LIN {X 0.076,Y -557.564,Z 1031.331,A 0.000,B 0.000,C 90.000,E1 95.625} C_DIS
LIN {X -0.086,Y -558.588,Z 1031.325,A 0.000,B 0.000,C 90.000,E1 94.531} C_DIS
LIN {X -0.162,Y -559.455,Z 1031.318,A 0.000,B 0.000,C 90.000,E1 93.151} C_DIS
LIN {X 0.192,Y -560.065,Z 1031.311,A 0.000,B 0.000,C 90.000,E1 92.007} C_DIS
LIN {X -0.259,Y -560.817,Z 1031.301,A 0.000,B 0.000,C 90.000,E1 90.115} C_DIS
LIN {X -0.131,Y -561.493,Z 1031.290,A 0.000,B 0.000,C 90.000,E1 88.165} C_DIS
LIN {X -0.179,Y -561.938,Z 1031.282,A 0.000,B 0.000,C 90.000,E1 86.788} C_DIS
LIN {X -0.001,Y -562.460,Z 1031.271,A 0.000,B 0.000,C 90.000,E1 84.837} C_DIS
LIN {X 0.054,Y -562.784,Z 1031.264,A 0.000,B 0.000,C 90.000,E1 83.451} C_DIS
LIN {X 0.026,Y -563.425,Z 1031.250,A 0.000,B 0.000,C 90.000,E1 80.971} C_DIS
LIN {X -0.056,Y -564.060,Z 1031.239,A 0.000,B 0.000,C 90.000,E1 79.050} C_DIS
LIN {X -0.009,Y -565.007,Z 1031.229,A 0.000,B 0.000,C 90.000,E1 77.117} C_DIS
LIN {X -0.145,Y -565.830,Z 1031.221,A 0.000,B 0.000,C 90.000,E1 75.755} C_DIS
LIN {X 0.008,Y -567.631,Z 1031.207,A 0.000,B 0.000,C 90.000,E1 73.268} C_DIS
LIN {X 0.206,Y -569.135,Z 1031.196,A 0.000,B 0.000,C 90.000,E1 71.329} C_DIS
LIN {X -0.249,Y -570.167,Z 1031.189,A 0.000,B 0.000,C 90.000,E1 70.007} C_DIS
LIN {X 0.058,Y -571.292,Z 1031.180,A 0.000,B 0.000,C 90.000,E1 68.337} C_DIS
LIN {X -0.147,Y -571.900,Z 1031.175,A 0.000,B 0.000,C 90.000,E1 67.539} C_DIS
LIN {X 0.029,Y -572.998,Z 1031.165,A 0.000,B 0.000,C 90.000,E1 65.613} C_DIS
LIN {X -0.261,Y -573.674,Z 1031.157,A 0.000,B 0.000,C 90.000,E1 64.280} C_DIS
LIN {X 0.073,Y -574.411,Z 1031.148,A 0.000,B 0.000,C 90.000,E1 62.615} C_DIS
LIN {X -0.093,Y -575.051,Z 1031.139,A 0.000,B 0.000,C 90.000,E1 61.001} C_DIS
LIN {X 0.182,Y -575.549,Z 1031.131,A 0.000,B 0.000,C 90.000,E1 59.616} C_DIS
LIN {X 0.132,Y -575.890,Z 1031.125,A 0.000,B 0.000,C 90.000,E1 58.535} C_DIS
LIN {X 0.236,Y -576.338,Z 1031.118,A 0.000,B 0.000,C 90.000,E1 57.168} C_DIS
LIN {X 0.200,Y -576.630,Z 1031.112,A 0.000,B 0.000,C 90.000,E1 56.087} C_DIS
LIN {X 0.011,Y -576.819,Z 1031.106,A 0.000,B 0.000,C 90.000,E1 55.022} C_DIS
LIN {X -0.194,Y -576.785,Z 1031.097,A 0.000,B 0.000,C 90.000,E1 53.417} C_DIS
LIN {X 0.128,Y -576.651,Z 1031.089,A 0.000,B 0.000,C 90.000,E1 52.029} C_DIS
LIN {X -0.218,Y -576.391,Z 1031.085,A 0.000,B 0.000,C 90.000,E1 51.251} C_DIS
LIN {X -0.206,Y -575.560,Z 1031.076,A 0.000,B 0.000,C 90.000,E1 49.622} C_DIS
LIN {X 0.016,Y -574.718,Z 1031.068,A 0.000,B 0.000,C 90.000,E1 48.243} C_DIS
LIN {X 0.093,Y -573.759,Z 1031.062,A 0.000,B 0.000,C 90.000,E1 47.148} C_DIS
LIN {X 0.034,Y -572.953,Z 1031.057,A 0.000,B 0.000,C 90.000,E1 46.338} C_DIS
LIN {X -0.137,Y -572.374,Z 1031.054,A 0.000,B 0.000,C 90.000,E1 45.810} C_DIS
LIN {X 0.302,Y -570.759,Z 1031.048,A 0.000,B 0.000,C 90.000,E1 44.676} C_DIS
LIN {X 0.211,Y -569.409,Z 1031.044,A 0.000,B 0.000,C 90.000,E1 43.866} C_DIS
LIN {X 0.211,Y -567.408,Z 1031.038,A 0.000,B 0.000,C 90.000,E1 42.771} C_DIS
LIN {X 0.075,Y -565.690,Z 1031.033,A 0.000,B 0.000,C 90.000,E1 41.962} C_DIS
LIN {X -0.036,Y -563.699,Z 1031.029,A 0.000,B 0.000,C 90.000,E1 41.148} C_DIS
LIN {X 0.299,Y -560.686,Z 1031.022,A 0.000,B 0.000,C 90.000,E1 40.011} C_DIS
LIN {X 0.143,Y -558.060,Z 1031.018,A 0.000,B 0.000,C 90.000,E1 39.197} C_DIS
LIN {X -0.040,Y -555.136,Z 1031.013,A 0.000,B 0.000,C 90.000,E1 38.382} C_DIS
LIN {X 0.112,Y -553.067,Z 1031.010,A 0.000,B 0.000,C 90.000,E1 37.810} C_DIS
LIN {X -0.126,Y -549.576,Z 1031.005,A 0.000,B 0.000,C 90.000,E1 36.996} C_DIS
LIN {X -0.107,Y -545.200,Z 1031.000,A 0.000,B 0.000,C 90.000,E1 36.011} C_DIS
LIN {X -0.144,Y -540.444,Z 1030.995,A 0.000,B 0.000,C 90.000,E1 35.025} C_DIS
LIN {X 0.198,Y -535.208,Z 1030.989,A 0.000,B 0.000,C 90.000,E1 33.992} C_DIS
LIN {X -0.111,Y -530.442,Z 1030.984,A 0.000,B 0.000,C 90.000,E1 33.166} C_DIS
LIN {X 0.133,Y -526.175,Z 1030.980,A 0.000,B 0.000,C 90.000,E1 32.418} C_DIS
LIN {X -0.223,Y -522.546,Z 1030.977,A 0.000,B 0.000,C 90.000,E1 31.878} C_DIS
LIN {X 0.112,Y -518.686,Z 1030.974,A 0.000,B 0.000,C 90.000,E1 31.258} C_DIS
LIN {X 0.146,Y -514.647,Z 1030.971,A 0.000,B 0.000,C 90.000,E1 30.669} C_DIS
LIN {X 0.154,Y -510.295,Z 1030.967,A 0.000,B 0.000,C 90.000,E1 30.079} C_DIS
LIN {X 0.195,Y -504.310,Z 1030.963,A 0.000,B 0.000,C 90.000,E1 29.333} C_DIS
LIN {X 0.071,Y -498.036,Z 1030.959,A 0.000,B 0.000,C 90.000,E1 28.615} C_DIS
LIN {X 0.036,Y -491.414,Z 1030.955,A 0.000,B 0.000,C 90.000,E1 27.897} C_DIS
LIN {X -0.129,Y -481.583,Z 1030.950,A 0.000,B 0.000,C 90.000,E1 26.924} C_DIS
LIN {X -0.074,Y -473.013,Z 1030.945,A 0.000,B 0.000,C 90.000,E1 26.104} C_DIS
LIN {X 0.009,Y -465.593,Z 1030.941,A 0.000,B 0.000,C 90.000,E1 25.412} C_DIS
LIN {X -0.083,Y -459.799,Z 1030.938,A 0.000,B 0.000,C 90.000,E1 24.899} C_DIS
LIN {X 0.065,Y -446.062,Z 1030.932,A 0.000,B 0.000,C 90.000,E1 23.718} C_DIS
LIN {X 0.224,Y -433.951,Z 1030.926,A 0.000,B 0.000,C 90.000,E1 22.642} C_DIS
LIN {X 0.260,Y -416.687,Z 1030.917,A 0.000,B 0.000,C 90.000,E1 20.972} C_DIS
LIN {X 0.130,Y -404.180,Z 1030.909,A 0.000,B 0.000,C 90.000,E1 19.631} C_DIS
LIN {X -0.123,Y -400.264,Z 1030.907,A 0.000,B 0.000,C 90.000,E1 19.195} C_DIS
LIN {X 0.180,Y -395.883,Z 1030.903,A 0.000,B 0.000,C 90.000,E1 18.544} C_DIS
LIN {X -0.083,Y -394.801,Z 1030.902,A 0.000,B 0.000,C 90.000,E1 18.417} C_DIS
LIN {X -0.153,Y -392.202,Z 1030.899,A 0.000,B 0.000,C 90.000,E1 17.819} C_DIS
LIN {X 0.040,Y -391.374,Z 1030.896,A 0.000,B 0.000,C 90.000,E1 17.347} C_DIS
LIN {X 0.136,Y -391.156,Z 1030.892,A 0.000,B 0.000,C 90.000,E1 16.622} C_DIS
LIN {X -0.134,Y -391.911,Z 1030.887,A 0.000,B 0.000,C 90.000,E1 15.607} C_DIS
LIN {X -0.095,Y -395.576,Z 1030.869,A 0.000,B 0.000,C 90.000,E1 12.411} C_DIS
LIN {X 0.093,Y -402.719,Z 1030.844,A 0.000,B 0.000,C 90.000,E1 7.814} C_DIS
LIN {X -0.033,Y -410.656,Z 1030.822,A 0.000,B 0.000,C 90.000,E1 4.012} C_DIS
LIN {X -0.055,Y -412.062,Z 1030.818,A 0.000,B 0.000,C 90.000,E1 3.326} C_DIS
LIN {X -0.035,Y -413.975,Z 1030.815,A 0.000,B 0.000,C 90.000,E1 2.636} C_DIS
LIN {X -0.033,Y -414.560,Z 1030.814,A 0.000,B 0.000,C 90.000,E1 2.465} C_DIS
LIN {X 0.192,Y -417.332,Z 1030.810,A 0.000,B 0.000,C 90.000,E1 1.835} C_DIS
LIN {X 0.009,Y -419.415,Z 1030.809,A 0.000,B 0.000,C 90.000,E1 1.604} C_DIS
LIN {X 0.152,Y -422.272,Z 1030.807,A 0.000,B 0.000,C 90.000,E1 1.260} C_DIS
LIN {X -0.175,Y -424.261,Z 1030.806,A 0.000,B 0.000,C 90.000,E1 1.146} C_DIS
LIN {X -0.084,Y -428.213,Z 1030.805,A 0.000,B 0.000,C 90.000,E1 0.859} C_DIS
LIN {X -0.182,Y -433.472,Z 1030.803,A 0.000,B 0.000,C 90.000,E1 0.573} C_DIS
LIN {X -0.208,Y -453.935,Z 1030.796,A 0.000,B 0.000,C 90.000,E1 359.312} C_DIS
LIN {X 0.128,Y -470.538,Z 1030.791,A 0.000,B 0.000,C 90.000,E1 358.282} C_DIS
LIN {X -0.068,Y -491.833,Z 1030.783,A 0.000,B 0.000,C 90.000,E1 357.020} C_DIS
LIN {X 0.105,Y -499.780,Z 1030.781,A 0.000,B 0.000,C 90.000,E1 356.502} C_DIS
LIN {X 0.166,Y -509.387,Z 1030.777,A 0.000,B 0.000,C 90.000,E1 355.869} C_DIS
LIN {X -0.108,Y -515.488,Z 1030.775,A 0.000,B 0.000,C 90.000,E1 355.469} C_DIS
LIN {X -0.001,Y -522.956,Z 1030.772,A 0.000,B 0.000,C 90.000,E1 354.894} C_DIS
LIN {X -0.190,Y -530.141,Z 1030.768,A 0.000,B 0.000,C 90.000,E1 354.318} C_DIS
LIN {X -0.119,Y -537.076,Z 1030.765,A 0.000,B 0.000,C 90.000,E1 353.685} C_DIS
LIN {X -0.152,Y -542.491,Z 1030.762,A 0.000,B 0.000,C 90.000,E1 353.166} C_DIS
LIN {X 0.060,Y -548.742,Z 1030.758,A 0.000,B 0.000,C 90.000,E1 352.470} C_DIS
LIN {X -0.019,Y -554.412,Z 1030.754,A 0.000,B 0.000,C 90.000,E1 351.781} C_DIS
LIN {X -0.152,Y -557.710,Z 1030.752,A 0.000,B 0.000,C 90.000,E1 351.376} C_DIS
LIN {X 0.273,Y -563.373,Z 1030.747,A 0.000,B 0.000,C 90.000,E1 350.500} C_DIS
LIN {X -0.057,Y -566.861,Z 1030.744,A 0.000,B 0.000,C 90.000,E1 349.982} C_DIS
LIN {X 0.050,Y -570.878,Z 1030.741,A 0.000,B 0.000,C 90.000,E1 349.285} C_DIS
LIN {X -0.069,Y -573.900,Z 1030.738,A 0.000,B 0.000,C 90.000,E1 348.757} C_DIS
LIN {X -0.230,Y -576.728,Z 1030.734,A 0.000,B 0.000,C 90.000,E1 348.229} C_DIS
LIN {X -0.151,Y -580.588,Z 1030.730,A 0.000,B 0.000,C 90.000,E1 347.409} C_DIS
LIN {X -0.032,Y -584.307,Z 1030.726,A 0.000,B 0.000,C 90.000,E1 346.589} C_DIS
LIN {X -0.060,Y -588.917,Z 1030.720,A 0.000,B 0.000,C 90.000,E1 345.519} C_DIS
LIN {X 0.247,Y -594.335,Z 1030.712,A 0.000,B 0.000,C 90.000,E1 344.157} C_DIS
LIN {X 0.083,Y -597.476,Z 1030.708,A 0.000,B 0.000,C 90.000,E1 343.378} C_DIS
LIN {X 0.237,Y -601.515,Z 1030.702,A 0.000,B 0.000,C 90.000,E1 342.308} C_DIS
LIN {X -0.225,Y -606.144,Z 1030.695,A 0.000,B 0.000,C 90.000,E1 341.040} C_DIS
LIN {X -0.075,Y -608.728,Z 1030.690,A 0.000,B 0.000,C 90.000,E1 340.242} C_DIS
LIN {X -0.161,Y -611.891,Z 1030.684,A 0.000,B 0.000,C 90.000,E1 339.209} C_DIS
LIN {X -0.284,Y -616.270,Z 1030.676,A 0.000,B 0.000,C 90.000,E1 337.667} C_DIS
LIN {X -0.077,Y -620.163,Z 1030.667,A 0.000,B 0.000,C 90.000,E1 336.102} C_DIS
LIN {X 0.207,Y -623.072,Z 1030.660,A 0.000,B 0.000,C 90.000,E1 334.793} C_DIS
LIN {X 0.236,Y -625.574,Z 1030.653,A 0.000,B 0.000,C 90.000,E1 333.512} C_DIS
LIN {X -0.247,Y -627.895,Z 1030.646,A 0.000,B 0.000,C 90.000,E1 332.281} C_DIS
LIN {X -0.145,Y -629.803,Z 1030.639,A 0.000,B 0.000,C 90.000,E1 331.001} C_DIS
LIN {X 0.082,Y -631.838,Z 1030.630,A 0.000,B 0.000,C 90.000,E1 329.459} C_DIS
LIN {X -0.001,Y -633.183,Z 1030.623,A 0.000,B 0.000,C 90.000,E1 328.201} C_DIS
LIN {X 0.267,Y -634.278,Z 1030.616,A 0.000,B 0.000,C 90.000,E1 326.914} C_DIS
LIN {X 0.019,Y -635.199,Z 1030.609,A 0.000,B 0.000,C 90.000,E1 325.674} C_DIS
LIN {X -0.234,Y -635.607,Z 1030.604,A 0.000,B 0.000,C 90.000,E1 324.689} C_DIS
LIN {X 0.032,Y -635.908,Z 1030.598,A 0.000,B 0.000,C 90.000,E1 323.657} C_DIS
LIN {X -0.083,Y -636.106,Z 1030.588,A 0.000,B 0.000,C 90.000,E1 321.904} C_DIS
LIN {X -0.291,Y -636.618,Z 1030.577,A 0.000,B 0.000,C 90.000,E1 319.908} C_DIS
LIN {X 0.015,Y -637.127,Z 1030.567,A 0.000,B 0.000,C 90.000,E1 318.119} C_DIS
LIN {X -0.194,Y -637.527,Z 1030.558,A 0.000,B 0.000,C 90.000,E1 316.377} C_DIS
LIN {X 0.154,Y -638.045,Z 1030.549,A 0.000,B 0.000,C 90.000,E1 314.838} C_DIS
LIN {X -0.108,Y -638.830,Z 1030.538,A 0.000,B 0.000,C 90.000,E1 312.852} C_DIS
LIN {X -0.093,Y -639.157,Z 1030.531,A 0.000,B 0.000,C 90.000,E1 311.595} C_DIS
LIN {X -0.015,Y -639.485,Z 1030.524,A 0.000,B 0.000,C 90.000,E1 310.334} C_DIS
LIN {X -0.024,Y -639.739,Z 1030.516,A 0.000,B 0.000,C 90.000,E1 308.830} C_DIS
LIN {X 0.070,Y -639.862,Z 1030.507,A 0.000,B 0.000,C 90.000,E1 307.317} C_DIS
LIN {X -0.421,Y -640.311,Z 1030.495,A 0.000,B 0.000,C 90.000,E1 305.105} C_DIS
LIN {X 0.229,Y -640.938,Z 1030.485,A 0.000,B 0.000,C 90.000,E1 303.293} C_DIS
LIN {X -0.205,Y -643.073,Z 1030.467,A 0.000,B 0.000,C 90.000,E1 300.079} C_DIS
LIN {X -0.168,Y -643.943,Z 1030.462,A 0.000,B 0.000,C 90.000,E1 299.077} C_DIS
LIN {X -0.201,Y -645.660,Z 1030.452,A 0.000,B 0.000,C 90.000,E1 297.334} C_DIS
LIN {X 0.131,Y -646.493,Z 1030.446,A 0.000,B 0.000,C 90.000,E1 296.309} C_DIS
LIN {X -0.197,Y -647.035,Z 1030.442,A 0.000,B 0.000,C 90.000,E1 295.591} C_DIS
LIN {X -0.129,Y -647.348,Z 1030.437,A 0.000,B 0.000,C 90.000,E1 294.591} C_DIS
LIN {X -0.049,Y -647.402,Z 1030.431,A 0.000,B 0.000,C 90.000,E1 293.590} C_DIS
LIN {X 0.199,Y -647.185,Z 1030.427,A 0.000,B 0.000,C 90.000,E1 292.823} C_DIS
LIN {X 0.186,Y -647.001,Z 1030.423,A 0.000,B 0.000,C 90.000,E1 292.078} C_DIS
LIN {X 0.097,Y -646.531,Z 1030.420,A 0.000,B 0.000,C 90.000,E1 291.589} C_DIS
LIN {X -0.066,Y -646.206,Z 1030.419,A 0.000,B 0.000,C 90.000,E1 291.354} C_DIS
LIN {X 0.075,Y -645.233,Z 1030.416,A 0.000,B 0.000,C 90.000,E1 290.844} C_DIS
LIN {X -0.087,Y -644.328,Z 1030.415,A 0.000,B 0.000,C 90.000,E1 290.610} C_DIS
LIN {X -0.218,Y -642.726,Z 1030.412,A 0.000,B 0.000,C 90.000,E1 290.248} C_DIS
LIN {X -0.188,Y -642.028,Z 1030.412,A 0.000,B 0.000,C 90.000,E1 290.120} C_DIS
LIN {X -0.135,Y -639.828,Z 1030.410,A 0.000,B 0.000,C 90.000,E1 289.866} C_DIS
LIN {X 0.314,Y -636.233,Z 1030.408,A 0.000,B 0.000,C 90.000,E1 289.450} C_DIS
LIN {X 0.120,Y -634.358,Z 1030.408,A 0.000,B 0.000,C 90.000,E1 289.341} C_DIS
LIN {X 0.139,Y -630.829,Z 1030.406,A 0.000,B 0.000,C 90.000,E1 289.141} C_DIS
LIN {X 0.196,Y -628.129,Z 1030.406,A 0.000,B 0.000,C 90.000,E1 288.960} C_DIS
LIN {X -0.171,Y -622.192,Z 1030.404,A 0.000,B 0.000,C 90.000,E1 288.725} C_DIS
LIN {X 0.100,Y -615.171,Z 1030.402,A 0.000,B 0.000,C 90.000,E1 288.417} C_DIS
LIN {X -0.135,Y -602.825,Z 1030.400,A 0.000,B 0.000,C 90.000,E1 288.000} C_DIS
LIN {X 0.000,Y -599.579,Z 1030.399,A 0.000,B 0.000,C 90.000,E1 287.873} C_DIS
LIN {X -0.039,Y -599.565,Z 1030.399,A 0.000,B 0.000,C 90.000,E1 287.873} C_DIS
LIN {X -0.015,Y -599.723,Z 1030.398,A 0.000,B 0.000,C 90.000,E1 287.692} C_DIS
LIN {X 0.213,Y -600.694,Z 1030.398,A 0.000,B 0.000,C 90.000,E1 287.583} C_DIS
LIN {X 0.209,Y -604.492,Z 1030.396,A 0.000,B 0.000,C 90.000,E1 287.275} C_DIS
LIN {X 0.233,Y -609.715,Z 1030.394,A 0.000,B 0.000,C 90.000,E1 286.804} C_DIS
LIN {X 0.186,Y -611.990,Z 1030.392,A 0.000,B 0.000,C 90.000,E1 286.567} C_DIS
LIN {X -0.101,Y -615.474,Z 1030.390,A 0.000,B 0.000,C 90.000,E1 286.205} C_DIS
LIN {X -0.044,Y -620.583,Z 1030.386,A 0.000,B 0.000,C 90.000,E1 285.426} C_DIS
LIN {X 0.086,Y -624.017,Z 1030.382,A 0.000,B 0.000,C 90.000,E1 284.773} C_DIS
LIN {X 0.270,Y -626.266,Z 1030.379,A 0.000,B 0.000,C 90.000,E1 284.245} C_DIS
LIN {X 0.063,Y -627.301,Z 1030.378,A 0.000,B 0.000,C 90.000,E1 284.008} C_DIS
LIN {X -0.340,Y -628.912,Z 1030.375,A 0.000,B 0.000,C 90.000,E1 283.536} C_DIS
LIN {X -0.313,Y -630.598,Z 1030.371,A 0.000,B 0.000,C 90.000,E1 282.771} C_DIS
LIN {X -0.080,Y -631.239,Z 1030.368,A 0.000,B 0.000,C 90.000,E1 282.243} C_DIS
LIN {X -0.270,Y -631.307,Z 1030.367,A 0.000,B 0.000,C 90.000,E1 282.007} C_DIS
LIN {X -0.032,Y -631.110,Z 1030.364,A 0.000,B 0.000,C 90.000,E1 281.478} C_DIS
LIN {X 0.203,Y -630.530,Z 1030.361,A 0.000,B 0.000,C 90.000,E1 280.950} C_DIS
LIN {X -0.302,Y -629.473,Z 1030.358,A 0.000,B 0.000,C 90.000,E1 280.489} C_DIS
LIN {X 0.122,Y -628.763,Z 1030.357,A 0.000,B 0.000,C 90.000,E1 280.197} C_DIS
LIN {X 0.337,Y -626.967,Z 1030.354,A 0.000,B 0.000,C 90.000,E1 279.670} C_DIS
LIN {X -0.180,Y -624.785,Z 1030.351,A 0.000,B 0.000,C 90.000,E1 279.208} C_DIS
LIN {X 0.001,Y -621.439,Z 1030.348,A 0.000,B 0.000,C 90.000,E1 278.681} C_DIS
LIN {X 0.061,Y -617.619,Z 1030.345,A 0.000,B 0.000,C 90.000,E1 278.163} C_DIS
LIN {X -0.101,Y -616.554,Z 1030.345,A 0.000,B 0.000,C 90.000,E1 278.049} C_DIS
LIN {X 0.145,Y -611.575,Z 1030.342,A 0.000,B 0.000,C 90.000,E1 277.530} C_DIS
LIN {X 0.115,Y -607.533,Z 1030.340,A 0.000,B 0.000,C 90.000,E1 277.182} C_DIS
LIN {X 0.238,Y -603.028,Z 1030.338,A 0.000,B 0.000,C 90.000,E1 276.834} C_DIS
LIN {X -0.104,Y -598.455,Z 1030.336,A 0.000,B 0.000,C 90.000,E1 276.549} C_DIS
LIN {X -0.163,Y -593.446,Z 1030.335,A 0.000,B 0.000,C 90.000,E1 276.258} C_DIS
LIN {X 0.279,Y -588.823,Z 1030.333,A 0.000,B 0.000,C 90.000,E1 275.967} C_DIS
LIN {X -0.045,Y -586.868,Z 1030.333,A 0.000,B 0.000,C 90.000,E1 275.910} C_DIS
LIN {X 0.252,Y -580.426,Z 1030.332,A 0.000,B 0.000,C 90.000,E1 275.682} C_DIS
LIN {X -0.055,Y -573.670,Z 1030.331,A 0.000,B 0.000,C 90.000,E1 275.568} C_DIS
LIN {X -0.222,Y -566.832,Z 1030.331,A 0.000,B 0.000,C 90.000,E1 275.511} C_DIS
LIN {X -0.241,Y -543.919,Z 1030.331,A 0.000,B 0.000,C 90.000,E1 275.511} C_DIS
LIN {X -0.040,Y -543.531,Z 1030.330,A 0.000,B 0.000,C 90.000,E1 275.391} C_DIS
LIN {X 0.132,Y -543.095,Z 1030.328,A 0.000,B 0.000,C 90.000,E1 275.106} C_DIS
LIN {X -0.125,Y -542.527,Z 1030.325,A 0.000,B 0.000,C 90.000,E1 274.588} C_DIS
LIN {X -0.104,Y -542.123,Z 1030.324,A 0.000,B 0.000,C 90.000,E1 274.302} C_DIS
LIN {X 0.231,Y -540.064,Z 1030.305,A 0.000,B 0.000,C 90.000,E1 270.859} C_DIS
LIN {X -0.231,Y -539.398,Z 1030.299,A 0.000,B 0.000,C 90.000,E1 269.771} C_DIS
LIN {X -0.122,Y -538.177,Z 1030.289,A 0.000,B 0.000,C 90.000,E1 268.051} C_DIS
LIN {X -0.046,Y -537.093,Z 1030.281,A 0.000,B 0.000,C 90.000,E1 266.617} C_DIS
LIN {X 0.074,Y -535.412,Z 1030.269,A 0.000,B 0.000,C 90.000,E1 264.318} C_DIS
LIN {X 0.182,Y -534.307,Z 1030.261,A 0.000,B 0.000,C 90.000,E1 262.875} C_DIS
LIN {X 0.221,Y -533.225,Z 1030.254,A 0.000,B 0.000,C 90.000,E1 261.724} C_DIS
LIN {X -0.171,Y -532.274,Z 1030.249,A 0.000,B 0.000,C 90.000,E1 260.905} C_DIS
LIN {X 0.067,Y -529.662,Z 1030.237,A 0.000,B 0.000,C 90.000,E1 258.578} C_DIS
LIN {X 0.233,Y -528.179,Z 1030.229,A 0.000,B 0.000,C 90.000,E1 257.117} C_DIS
LIN {X 0.143,Y -525.955,Z 1030.217,A 0.000,B 0.000,C 90.000,E1 255.102} C_DIS
LIN {X 0.149,Y -523.431,Z 1030.204,A 0.000,B 0.000,C 90.000,E1 252.779} C_DIS
LIN {X 0.100,Y -521.875,Z 1030.196,A 0.000,B 0.000,C 90.000,E1 251.329} C_DIS
LIN {X 0.168,Y -519.656,Z 1030.187,A 0.000,B 0.000,C 90.000,E1 249.571} C_DIS
LIN {X -0.120,Y -517.331,Z 1030.177,A 0.000,B 0.000,C 90.000,E1 247.847} C_DIS
LIN {X 0.080,Y -515.408,Z 1030.169,A 0.000,B 0.000,C 90.000,E1 246.357} C_DIS
LIN {X -0.008,Y -514.200,Z 1030.164,A 0.000,B 0.000,C 90.000,E1 245.485} C_DIS
LIN {X -0.129,Y -511.916,Z 1030.156,A 0.000,B 0.000,C 90.000,E1 244.024} C_DIS
LIN {X -0.060,Y -509.524,Z 1030.147,A 0.000,B 0.000,C 90.000,E1 242.538} C_DIS
LIN {X -0.036,Y -506.959,Z 1030.139,A 0.000,B 0.000,C 90.000,E1 241.051} C_DIS
LIN {X 0.059,Y -503.785,Z 1030.129,A 0.000,B 0.000,C 90.000,E1 239.253} C_DIS
LIN {X -0.218,Y -501.005,Z 1030.121,A 0.000,B 0.000,C 90.000,E1 237.788} C_DIS
LIN {X 0.119,Y -498.597,Z 1030.114,A 0.000,B 0.000,C 90.000,E1 236.548} C_DIS
LIN {X -0.272,Y -496.091,Z 1030.108,A 0.000,B 0.000,C 90.000,E1 235.388} C_DIS
LIN {X -0.020,Y -493.358,Z 1030.101,A 0.000,B 0.000,C 90.000,E1 234.149} C_DIS
LIN {X 0.075,Y -490.507,Z 1030.094,A 0.000,B 0.000,C 90.000,E1 232.924} C_DIS
LIN {X -0.036,Y -486.918,Z 1030.086,A 0.000,B 0.000,C 90.000,E1 231.412} C_DIS
LIN {X 0.153,Y -481.359,Z 1030.072,A 0.000,B 0.000,C 90.000,E1 228.933} C_DIS
LIN {X 0.235,Y -477.296,Z 1030.062,A 0.000,B 0.000,C 90.000,E1 227.067} C_DIS
LIN {X 0.078,Y -472.113,Z 1030.048,A 0.000,B 0.000,C 90.000,E1 224.595} C_DIS
LIN {X 0.026,Y -470.139,Z 1030.043,A 0.000,B 0.000,C 90.000,E1 223.662} C_DIS
LIN {X 0.108,Y -466.933,Z 1030.034,A 0.000,B 0.000,C 90.000,E1 222.081} C_DIS
LIN {X -0.192,Y -463.713,Z 1030.025,A 0.000,B 0.000,C 90.000,E1 220.539} C_DIS
LIN {X 0.152,Y -460.400,Z 1030.016,A 0.000,B 0.000,C 90.000,E1 218.910} C_DIS
LIN {X 0.143,Y -456.795,Z 1030.007,A 0.000,B 0.000,C 90.000,E1 217.317} C_DIS
LIN {X -0.043,Y -451.241,Z 1029.993,A 0.000,B 0.000,C 90.000,E1 214.771} C_DIS
LIN {X -0.053,Y -447.112,Z 1029.982,A 0.000,B 0.000,C 90.000,E1 212.832} C_DIS
LIN {X -0.029,Y -442.831,Z 1029.972,A 0.000,B 0.000,C 90.000,E1 210.875} C_DIS
LIN {X 0.178,Y -439.976,Z 1029.964,A 0.000,B 0.000,C 90.000,E1 209.539} C_DIS
LIN {X 0.148,Y -436.205,Z 1029.955,A 0.000,B 0.000,C 90.000,E1 207.897} C_DIS
LIN {X 0.042,Y -431.677,Z 1029.944,A 0.000,B 0.000,C 90.000,E1 205.924} C_DIS
LIN {X 0.027,Y -426.499,Z 1029.931,A 0.000,B 0.000,C 90.000,E1 203.590} C_DIS
LIN {X -0.091,Y -422.343,Z 1029.920,A 0.000,B 0.000,C 90.000,E1 201.589} C_DIS
LIN {X -0.060,Y -417.873,Z 1029.907,A 0.000,B 0.000,C 90.000,E1 199.214} C_DIS
LIN {X 0.001,Y -412.870,Z 1029.890,A 0.000,B 0.000,C 90.000,E1 196.134} C_DIS
LIN {X -0.056,Y -408.713,Z 1029.871,A 0.000,B 0.000,C 90.000,E1 192.703} C_DIS
LIN {X 0.001,Y -408.004,Z 1029.865,A 0.000,B 0.000,C 90.000,E1 191.658} C_DIS
LIN {X 0.118,Y -407.805,Z 1029.861,A 0.000,B 0.000,C 90.000,E1 190.950} C_DIS
LIN {X 0.136,Y -407.876,Z 1029.859,A 0.000,B 0.000,C 90.000,E1 190.602} C_DIS
LIN {X 0.154,Y -408.167,Z 1029.857,A 0.000,B 0.000,C 90.000,E1 190.254} C_DIS
LIN {X 0.172,Y -408.634,Z 1029.855,A 0.000,B 0.000,C 90.000,E1 189.905} C_DIS
LIN {X -0.084,Y -410.388,Z 1029.851,A 0.000,B 0.000,C 90.000,E1 189.265} C_DIS
LIN {X -0.059,Y -411.723,Z 1029.849,A 0.000,B 0.000,C 90.000,E1 188.916} C_DIS
LIN {X 0.031,Y -414.879,Z 1029.846,A 0.000,B 0.000,C 90.000,E1 188.276} C_DIS
LIN {X -0.082,Y -420.138,Z 1029.841,A 0.000,B 0.000,C 90.000,E1 187.466} C_DIS
LIN {X -0.040,Y -433.626,Z 1029.832,A 0.000,B 0.000,C 90.000,E1 185.682} C_DIS
LIN {X -0.229,Y -439.930,Z 1029.827,A 0.000,B 0.000,C 90.000,E1 184.878} C_DIS
LIN {X 0.023,Y -445.056,Z 1029.823,A 0.000,B 0.000,C 90.000,E1 184.188} C_DIS
LIN {X -0.192,Y -452.309,Z 1029.818,A 0.000,B 0.000,C 90.000,E1 183.269} C_DIS
LIN {X -0.204,Y -458.528,Z 1029.814,A 0.000,B 0.000,C 90.000,E1 182.465} C_DIS
LIN {X -0.099,Y -468.019,Z 1029.807,A 0.000,B 0.000,C 90.000,E1 181.203} C_DIS
LIN {X 0.014,Y -474.515,Z 1029.802,A 0.000,B 0.000,C 90.000,E1 180.286} C_DIS
LIN {X -0.131,Y -481.002,Z 1029.797,A 0.000,B 0.000,C 90.000,E1 179.370} C_DIS
LIN {X -0.209,Y -487.392,Z 1029.791,A 0.000,B 0.000,C 90.000,E1 178.453} C_DIS
LIN {X -0.148,Y -493.622,Z 1029.786,A 0.000,B 0.000,C 90.000,E1 177.535} C_DIS
LIN {X 0.129,Y -500.432,Z 1029.780,A 0.000,B 0.000,C 90.000,E1 176.445} C_DIS
LIN {X 0.181,Y -507.917,Z 1029.774,A 0.000,B 0.000,C 90.000,E1 175.241} C_DIS
LIN {X -0.216,Y -512.253,Z 1029.770,A 0.000,B 0.000,C 90.000,E1 174.546} C_DIS
LIN {X 0.199,Y -514.267,Z 1029.768,A 0.000,B 0.000,C 90.000,E1 174.204} C_DIS
LIN {X 0.041,Y -524.353,Z 1029.758,A 0.000,B 0.000,C 90.000,E1 172.470} C_DIS
LIN {X 0.248,Y -530.202,Z 1029.753,A 0.000,B 0.000,C 90.000,E1 171.432} C_DIS
LIN {X 0.135,Y -537.511,Z 1029.745,A 0.000,B 0.000,C 90.000,E1 170.151} C_DIS
LIN {X 0.146,Y -544.826,Z 1029.738,A 0.000,B 0.000,C 90.000,E1 168.870} C_DIS
LIN {X 0.002,Y -551.184,Z 1029.732,A 0.000,B 0.000,C 90.000,E1 167.757} C_DIS
LIN {X 0.213,Y -556.502,Z 1029.727,A 0.000,B 0.000,C 90.000,E1 166.756} C_DIS
LIN {X 0.100,Y -563.101,Z 1029.720,A 0.000,B 0.000,C 90.000,E1 165.519} C_DIS
LIN {X 0.080,Y -569.639,Z 1029.713,A 0.000,B 0.000,C 90.000,E1 164.283} C_DIS
LIN {X 0.213,Y -576.549,Z 1029.705,A 0.000,B 0.000,C 90.000,E1 162.906} C_DIS
LIN {X 0.140,Y -579.776,Z 1029.701,A 0.000,B 0.000,C 90.000,E1 162.236} C_DIS
LIN {X 0.312,Y -584.117,Z 1029.696,A 0.000,B 0.000,C 90.000,E1 161.275} C_DIS
LIN {X -0.096,Y -588.684,Z 1029.690,A 0.000,B 0.000,C 90.000,E1 160.242} C_DIS
LIN {X 0.105,Y -593.091,Z 1029.684,A 0.000,B 0.000,C 90.000,E1 159.156} C_DIS
LIN {X 0.020,Y -597.247,Z 1029.678,A 0.000,B 0.000,C 90.000,E1 158.103} C_DIS
LIN {X 0.076,Y -600.132,Z 1029.674,A 0.000,B 0.000,C 90.000,E1 157.305} C_DIS
LIN {X 0.328,Y -603.773,Z 1029.668,A 0.000,B 0.000,C 90.000,E1 156.230} C_DIS
LIN {X -0.216,Y -607.938,Z 1029.661,A 0.000,B 0.000,C 90.000,E1 154.973} C_DIS
LIN {X 0.152,Y -611.023,Z 1029.655,A 0.000,B 0.000,C 90.000,E1 153.896} C_DIS
LIN {X 0.045,Y -613.271,Z 1029.651,A 0.000,B 0.000,C 90.000,E1 153.127} C_DIS
LIN {X -0.066,Y -615.986,Z 1029.645,A 0.000,B 0.000,C 90.000,E1 152.103} C_DIS
LIN {X 0.119,Y -620.004,Z 1029.636,A 0.000,B 0.000,C 90.000,E1 150.539} C_DIS
LIN {X 0.155,Y -624.576,Z 1029.626,A 0.000,B 0.000,C 90.000,E1 148.742} C_DIS
LIN {X 0.100,Y -628.842,Z 1029.617,A 0.000,B 0.000,C 90.000,E1 146.962} C_DIS
LIN {X -0.064,Y -630.706,Z 1029.612,A 0.000,B 0.000,C 90.000,E1 146.215} C_DIS
LIN {X 0.008,Y -634.368,Z 1029.604,A 0.000,B 0.000,C 90.000,E1 144.689} C_DIS
LIN {X 0.011,Y -637.940,Z 1029.595,A 0.000,B 0.000,C 90.000,E1 143.176} C_DIS
LIN {X 0.093,Y -641.521,Z 1029.587,A 0.000,B 0.000,C 90.000,E1 141.662} C_DIS
LIN {X -0.180,Y -644.509,Z 1029.580,A 0.000,B 0.000,C 90.000,E1 140.436} C_DIS
LIN {X -0.143,Y -648.573,Z 1029.570,A 0.000,B 0.000,C 90.000,E1 138.690} C_DIS
LIN {X -0.155,Y -654.635,Z 1029.557,A 0.000,B 0.000,C 90.000,E1 136.215} C_DIS
LIN {X -0.443,Y -660.609,Z 1029.544,A 0.000,B 0.000,C 90.000,E1 134.028} C_DIS
LIN {X -0.071,Y -665.626,Z 1029.535,A 0.000,B 0.000,C 90.000,E1 132.285} C_DIS
LIN {X -0.041,Y -668.538,Z 1029.530,A 0.000,B 0.000,C 90.000,E1 131.310} C_DIS
LIN {X 0.039,Y -672.067,Z 1029.523,A 0.000,B 0.000,C 90.000,E1 130.092} C_DIS
LIN {X -0.249,Y -676.069,Z 1029.515,A 0.000,B 0.000,C 90.000,E1 128.669} C_DIS
LIN {X 0.030,Y -678.639,Z 1029.509,A 0.000,B 0.000,C 90.000,E1 127.684} C_DIS
LIN {X -0.172,Y -681.816,Z 1029.503,A 0.000,B 0.000,C 90.000,E1 126.503} C_DIS
LIN {X 0.388,Y -685.582,Z 1029.495,A 0.000,B 0.000,C 90.000,E1 125.025} C_DIS
LIN {X 0.065,Y -689.229,Z 1029.487,A 0.000,B 0.000,C 90.000,E1 123.627} C_DIS
LIN {X 0.003,Y -692.766,Z 1029.479,A 0.000,B 0.000,C 90.000,E1 122.212} C_DIS
LIN {X 0.124,Y -695.062,Z 1029.474,A 0.000,B 0.000,C 90.000,E1 121.258} C_DIS
LIN {X 0.264,Y -696.613,Z 1029.470,A 0.000,B 0.000,C 90.000,E1 120.541} C_DIS
LIN {X 0.080,Y -698.381,Z 1029.465,A 0.000,B 0.000,C 90.000,E1 119.617} C_DIS
LIN {X -0.085,Y -699.794,Z 1029.459,A 0.000,B 0.000,C 90.000,E1 118.693} C_DIS
LIN {X 0.108,Y -700.722,Z 1029.456,A 0.000,B 0.000,C 90.000,E1 117.975} C_DIS
LIN {X -0.082,Y -701.897,Z 1029.449,A 0.000,B 0.000,C 90.000,E1 116.821} C_DIS
LIN {X 0.406,Y -702.759,Z 1029.444,A 0.000,B 0.000,C 90.000,E1 115.848} C_DIS
LIN {X -0.058,Y -703.650,Z 1029.437,A 0.000,B 0.000,C 90.000,E1 114.719} C_DIS
LIN {X -0.134,Y -703.595,Z 1029.435,A 0.000,B 0.000,C 90.000,E1 114.259} C_DIS
LIN {X -0.141,Y -703.411,Z 1029.433,A 0.000,B 0.000,C 90.000,E1 114.027} C_DIS
LIN {X -0.224,Y -702.474,Z 1029.431,A 0.000,B 0.000,C 90.000,E1 113.567} C_DIS
LIN {X -0.226,Y -701.583,Z 1029.430,A 0.000,B 0.000,C 90.000,E1 113.334} C_DIS
LIN {X 0.315,Y -698.925,Z 1029.427,A 0.000,B 0.000,C 90.000,E1 112.823} C_DIS
LIN {X 0.176,Y -698.009,Z 1029.426,A 0.000,B 0.000,C 90.000,E1 112.717} C_DIS
LIN {X -0.336,Y -696.645,Z 1029.426,A 0.000,B 0.000,C 90.000,E1 112.642} C_DIS
LIN {X 0.139,Y -690.023,Z 1029.423,A 0.000,B 0.000,C 90.000,E1 112.206} C_DIS
LIN {X -0.296,Y -687.958,Z 1029.423,A 0.000,B 0.000,C 90.000,E1 112.153} C_DIS
LIN {X 0.165,Y -685.244,Z 1029.422,A 0.000,B 0.000,C 90.000,E1 112.025} C_DIS
LIN {X 0.124,Y -682.328,Z 1029.422,A 0.000,B 0.000,C 90.000,E1 111.972} C_DIS
LIN {X -0.007,Y -675.501,Z 1029.422,A 0.000,B 0.000,C 90.000,E1 111.897} C_DIS
LIN {X -0.054,Y -612.835,Z 1029.422,A 0.000,B 0.000,C 90.000,E1 111.897} C_DIS
LIN {X 0.289,Y -609.555,Z 1029.421,A 0.000,B 0.000,C 90.000,E1 111.770} C_DIS
LIN {X 0.117,Y -604.065,Z 1029.420,A 0.000,B 0.000,C 90.000,E1 111.589} C_DIS
LIN {X 0.046,Y -597.685,Z 1029.418,A 0.000,B 0.000,C 90.000,E1 111.280} C_DIS
LIN {X 0.015,Y -592.017,Z 1029.416,A 0.000,B 0.000,C 90.000,E1 110.918} C_DIS
LIN {X -0.066,Y -587.800,Z 1029.415,A 0.000,B 0.000,C 90.000,E1 110.610} C_DIS
LIN {X -0.303,Y -577.496,Z 1029.410,A 0.000,B 0.000,C 90.000,E1 109.758} C_DIS
LIN {X 0.222,Y -569.858,Z 1029.406,A 0.000,B 0.000,C 90.000,E1 109.141} C_DIS
LIN {X 0.141,Y -561.442,Z 1029.404,A 0.000,B 0.000,C 90.000,E1 108.671} C_DIS
LIN {X -0.202,Y -554.779,Z 1029.402,A 0.000,B 0.000,C 90.000,E1 108.362} C_DIS
LIN {X 0.226,Y -549.676,Z 1029.400,A 0.000,B 0.000,C 90.000,E1 108.000} C_DIS
LIN {X 0.172,Y -548.139,Z 1029.399,A 0.000,B 0.000,C 90.000,E1 107.819} C_DIS
LIN {X 0.130,Y -548.118,Z 1029.399,A 0.000,B 0.000,C 90.000,E1 107.819} C_DIS
LIN {X -0.261,Y -547.755,Z 1029.398,A 0.000,B 0.000,C 90.000,E1 107.583} C_DIS
LIN {X -0.244,Y -548.788,Z 1029.384,A 0.000,B 0.000,C 90.000,E1 105.190} C_DIS
LIN {X 0.006,Y -550.539,Z 1029.369,A 0.000,B 0.000,C 90.000,E1 102.355} C_DIS
LIN {X 0.100,Y -553.554,Z 1029.352,A 0.000,B 0.000,C 90.000,E1 99.265} C_DIS
LIN {X 0.125,Y -555.429,Z 1029.342,A 0.000,B 0.000,C 90.000,E1 97.587} C_DIS
LIN {X 0.000,Y -556.707,Z 1029.336,A 0.000,B 0.000,C 90.000,E1 96.486} C_DIS
LIN {X -0.105,Y -558.104,Z 1029.328,A 0.000,B 0.000,C 90.000,E1 95.106} C_DIS
LIN {X 0.172,Y -558.751,Z 1029.324,A 0.000,B 0.000,C 90.000,E1 94.245} C_DIS
LIN {X 0.102,Y -559.600,Z 1029.316,A 0.000,B 0.000,C 90.000,E1 92.865} C_DIS
LIN {X -0.079,Y -560.149,Z 1029.310,A 0.000,B 0.000,C 90.000,E1 91.776} C_DIS
LIN {X -0.080,Y -560.811,Z 1029.301,A 0.000,B 0.000,C 90.000,E1 90.115} C_DIS
LIN {X 0.048,Y -561.487,Z 1029.290,A 0.000,B 0.000,C 90.000,E1 88.165} C_DIS
LIN {X 0.000,Y -561.934,Z 1029.282,A 0.000,B 0.000,C 90.000,E1 86.788} C_DIS
LIN {X 0.087,Y -562.353,Z 1029.273,A 0.000,B 0.000,C 90.000,E1 85.122} C_DIS
LIN {X 0.084,Y -562.700,Z 1029.265,A 0.000,B 0.000,C 90.000,E1 83.742} C_DIS
LIN {X 0.132,Y -563.303,Z 1029.252,A 0.000,B 0.000,C 90.000,E1 81.254} C_DIS
LIN {X -0.041,Y -563.930,Z 1029.241,A 0.000,B 0.000,C 90.000,E1 79.342} C_DIS
LIN {X 0.166,Y -564.966,Z 1029.229,A 0.000,B 0.000,C 90.000,E1 77.117} C_DIS
LIN {X 0.197,Y -565.967,Z 1029.219,A 0.000,B 0.000,C 90.000,E1 75.463} C_DIS
LIN {X -0.032,Y -567.801,Z 1029.206,A 0.000,B 0.000,C 90.000,E1 73.015} C_DIS
LIN {X -0.340,Y -569.084,Z 1029.197,A 0.000,B 0.000,C 90.000,E1 71.402} C_DIS
LIN {X 0.273,Y -570.309,Z 1029.187,A 0.000,B 0.000,C 90.000,E1 69.699} C_DIS
LIN {X 0.198,Y -571.612,Z 1029.177,A 0.000,B 0.000,C 90.000,E1 67.794} C_DIS
LIN {X 0.213,Y -572.075,Z 1029.172,A 0.000,B 0.000,C 90.000,E1 66.975} C_DIS
LIN {X 0.200,Y -572.895,Z 1029.165,A 0.000,B 0.000,C 90.000,E1 65.613} C_DIS
LIN {X -0.091,Y -573.565,Z 1029.157,A 0.000,B 0.000,C 90.000,E1 64.280} C_DIS
LIN {X 0.240,Y -574.287,Z 1029.148,A 0.000,B 0.000,C 90.000,E1 62.615} C_DIS
LIN {X 0.229,Y -574.843,Z 1029.141,A 0.000,B 0.000,C 90.000,E1 61.257} C_DIS
LIN {X 0.007,Y -575.334,Z 1029.133,A 0.000,B 0.000,C 90.000,E1 59.921} C_DIS
LIN {X 0.293,Y -575.764,Z 1029.125,A 0.000,B 0.000,C 90.000,E1 58.535} C_DIS
LIN {X 0.376,Y -576.387,Z 1029.115,A 0.000,B 0.000,C 90.000,E1 56.628} C_DIS
LIN {X -0.165,Y -576.657,Z 1029.106,A 0.000,B 0.000,C 90.000,E1 55.055} C_DIS
LIN {X -0.198,Y -576.654,Z 1029.098,A 0.000,B 0.000,C 90.000,E1 53.703} C_DIS
LIN {X -0.078,Y -576.473,Z 1029.089,A 0.000,B 0.000,C 90.000,E1 52.065} C_DIS
LIN {X -0.071,Y -576.185,Z 1029.085,A 0.000,B 0.000,C 90.000,E1 51.251} C_DIS
LIN {X -0.065,Y -575.359,Z 1029.076,A 0.000,B 0.000,C 90.000,E1 49.622} C_DIS
LIN {X 0.154,Y -574.478,Z 1029.068,A 0.000,B 0.000,C 90.000,E1 48.243} C_DIS
LIN {X 0.227,Y -573.515,Z 1029.062,A 0.000,B 0.000,C 90.000,E1 47.148} C_DIS
LIN {X -0.230,Y -572.681,Z 1029.058,A 0.000,B 0.000,C 90.000,E1 46.377} C_DIS
LIN {X -0.007,Y -572.094,Z 1029.055,A 0.000,B 0.000,C 90.000,E1 45.810} C_DIS
LIN {X 0.022,Y -570.455,Z 1029.048,A 0.000,B 0.000,C 90.000,E1 44.717} C_DIS
LIN {X 0.333,Y -569.076,Z 1029.044,A 0.000,B 0.000,C 90.000,E1 43.866} C_DIS
LIN {X 0.327,Y -567.054,Z 1029.038,A 0.000,B 0.000,C 90.000,E1 42.771} C_DIS
LIN {X 0.291,Y -564.638,Z 1029.032,A 0.000,B 0.000,C 90.000,E1 41.676} C_DIS
LIN {X 0.072,Y -563.282,Z 1029.029,A 0.000,B 0.000,C 90.000,E1 41.148} C_DIS
LIN {X 0.039,Y -560.222,Z 1029.023,A 0.000,B 0.000,C 90.000,E1 40.048} C_DIS
LIN {X 0.238,Y -557.527,Z 1029.018,A 0.000,B 0.000,C 90.000,E1 39.197} C_DIS
LIN {X -0.028,Y -555.630,Z 1029.015,A 0.000,B 0.000,C 90.000,E1 38.669} C_DIS
LIN {X 0.197,Y -552.450,Z 1029.010,A 0.000,B 0.000,C 90.000,E1 37.810} C_DIS
LIN {X -0.047,Y -548.926,Z 1029.006,A 0.000,B 0.000,C 90.000,E1 36.996} C_DIS
LIN {X -0.219,Y -545.173,Z 1029.001,A 0.000,B 0.000,C 90.000,E1 36.171} C_DIS
LIN {X -0.086,Y -539.691,Z 1028.995,A 0.000,B 0.000,C 90.000,E1 35.025} C_DIS
LIN {X 0.246,Y -534.427,Z 1028.989,A 0.000,B 0.000,C 90.000,E1 33.992} C_DIS
LIN {X -0.073,Y -529.628,Z 1028.984,A 0.000,B 0.000,C 90.000,E1 33.166} C_DIS
LIN {X 0.164,Y -525.350,Z 1028.980,A 0.000,B 0.000,C 90.000,E1 32.418} C_DIS
LIN {X -0.199,Y -521.703,Z 1028.977,A 0.000,B 0.000,C 90.000,E1 31.878} C_DIS
LIN {X -0.039,Y -516.815,Z 1028.973,A 0.000,B 0.000,C 90.000,E1 31.131} C_DIS
LIN {X 0.071,Y -511.589,Z 1028.969,A 0.000,B 0.000,C 90.000,E1 30.384} C_DIS
LIN {X -0.129,Y -505.722,Z 1028.965,A 0.000,B 0.000,C 90.000,E1 29.667} C_DIS
LIN {X 0.065,Y -499.442,Z 1028.961,A 0.000,B 0.000,C 90.000,E1 28.899} C_DIS
LIN {X 0.128,Y -492.808,Z 1028.957,A 0.000,B 0.000,C 90.000,E1 28.153} C_DIS
LIN {X -0.025,Y -481.798,Z 1028.950,A 0.000,B 0.000,C 90.000,E1 27.052} C_DIS
LIN {X -0.024,Y -474.521,Z 1028.947,A 0.000,B 0.000,C 90.000,E1 26.360} C_DIS
LIN {X 0.053,Y -465.707,Z 1028.942,A 0.000,B 0.000,C 90.000,E1 25.540} C_DIS
LIN {X -0.170,Y -459.805,Z 1028.939,A 0.000,B 0.000,C 90.000,E1 25.027} C_DIS
LIN {X 0.085,Y -445.901,Z 1028.932,A 0.000,B 0.000,C 90.000,E1 23.823} C_DIS
LIN {X -0.118,Y -434.082,Z 1028.927,A 0.000,B 0.000,C 90.000,E1 22.823} C_DIS
LIN {X 0.126,Y -416.557,Z 1028.917,A 0.000,B 0.000,C 90.000,E1 21.099} C_DIS
LIN {X -0.036,Y -403.946,Z 1028.910,A 0.000,B 0.000,C 90.000,E1 19.758} C_DIS
LIN {X 0.128,Y -397.766,Z 1028.906,A 0.000,B 0.000,C 90.000,E1 18.960} C_DIS
LIN {X -0.121,Y -393.700,Z 1028.902,A 0.000,B 0.000,C 90.000,E1 18.362} C_DIS
LIN {X -0.057,Y -392.293,Z 1028.900,A 0.000,B 0.000,C 90.000,E1 18.000} C_DIS
LIN {X 0.021,Y -391.408,Z 1028.897,A 0.000,B 0.000,C 90.000,E1 17.457} C_DIS
LIN {X 0.046,Y -391.257,Z 1028.896,A 0.000,B 0.000,C 90.000,E1 17.275} C_DIS
LIN {X 0.116,Y -391.188,Z 1028.893,A 0.000,B 0.000,C 90.000,E1 16.732} C_DIS
LIN {X -0.214,Y -392.248,Z 1028.885,A 0.000,B 0.000,C 90.000,E1 15.371} C_DIS
LIN {X 0.223,Y -395.990,Z 1028.868,A 0.000,B 0.000,C 90.000,E1 12.119} C_DIS
LIN {X -0.015,Y -403.257,Z 1028.842,A 0.000,B 0.000,C 90.000,E1 7.587} C_DIS
LIN {X -0.122,Y -410.482,Z 1028.823,A 0.000,B 0.000,C 90.000,E1 4.131} C_DIS
LIN {X -0.100,Y -412.697,Z 1028.817,A 0.000,B 0.000,C 90.000,E1 3.094} C_DIS
LIN {X -0.103,Y -413.631,Z 1028.815,A 0.000,B 0.000,C 90.000,E1 2.751} C_DIS
LIN {X -0.099,Y -415.399,Z 1028.812,A 0.000,B 0.000,C 90.000,E1 2.236} C_DIS
LIN {X -0.089,Y -416.978,Z 1028.811,A 0.000,B 0.000,C 90.000,E1 1.892} C_DIS
LIN {X -0.068,Y -418.121,Z 1028.810,A 0.000,B 0.000,C 90.000,E1 1.718} C_DIS
LIN {X -0.014,Y -423.035,Z 1028.806,A 0.000,B 0.000,C 90.000,E1 1.146} C_DIS
LIN {X -0.153,Y -428.254,Z 1028.804,A 0.000,B 0.000,C 90.000,E1 0.802} C_DIS
LIN {X 0.116,Y -433.684,Z 1028.803,A 0.000,B 0.000,C 90.000,E1 0.458} C_DIS
LIN {X -0.212,Y -452.991,Z 1028.796,A 0.000,B 0.000,C 90.000,E1 359.312} C_DIS
LIN {X 0.122,Y -469.585,Z 1028.791,A 0.000,B 0.000,C 90.000,E1 358.282} C_DIS
LIN {X -0.025,Y -490.913,Z 1028.783,A 0.000,B 0.000,C 90.000,E1 357.020} C_DIS
LIN {X 0.145,Y -498.901,Z 1028.781,A 0.000,B 0.000,C 90.000,E1 356.502} C_DIS
LIN {X -0.148,Y -510.053,Z 1028.777,A 0.000,B 0.000,C 90.000,E1 355.812} C_DIS
LIN {X 0.152,Y -517.570,Z 1028.774,A 0.000,B 0.000,C 90.000,E1 355.241} C_DIS
LIN {X 0.209,Y -523.545,Z 1028.771,A 0.000,B 0.000,C 90.000,E1 354.780} C_DIS
LIN {X 0.118,Y -530.573,Z 1028.768,A 0.000,B 0.000,C 90.000,E1 354.204} C_DIS
LIN {X 0.164,Y -537.561,Z 1028.764,A 0.000,B 0.000,C 90.000,E1 353.571} C_DIS
LIN {X -0.220,Y -541.639,Z 1028.762,A 0.000,B 0.000,C 90.000,E1 353.223} C_DIS
LIN {X 0.206,Y -547.780,Z 1028.759,A 0.000,B 0.000,C 90.000,E1 352.534} C_DIS
LIN {X 0.192,Y -553.594,Z 1028.755,A 0.000,B 0.000,C 90.000,E1 351.837} C_DIS
LIN {X -0.115,Y -557.979,Z 1028.752,A 0.000,B 0.000,C 90.000,E1 351.310} C_DIS
LIN {X 0.228,Y -563.682,Z 1028.747,A 0.000,B 0.000,C 90.000,E1 350.443} C_DIS
LIN {X -0.102,Y -567.136,Z 1028.744,A 0.000,B 0.000,C 90.000,E1 349.926} C_DIS
LIN {X 0.305,Y -572.775,Z 1028.739,A 0.000,B 0.000,C 90.000,E1 348.926} C_DIS
LIN {X 0.231,Y -577.066,Z 1028.734,A 0.000,B 0.000,C 90.000,E1 348.117} C_DIS
LIN {X -0.253,Y -580.933,Z 1028.730,A 0.000,B 0.000,C 90.000,E1 347.353} C_DIS
LIN {X -0.231,Y -585.250,Z 1028.724,A 0.000,B 0.000,C 90.000,E1 346.408} C_DIS
LIN {X 0.326,Y -589.841,Z 1028.719,A 0.000,B 0.000,C 90.000,E1 345.283} C_DIS
LIN {X 0.080,Y -595.259,Z 1028.711,A 0.000,B 0.000,C 90.000,E1 343.976} C_DIS
LIN {X -0.074,Y -598.404,Z 1028.707,A 0.000,B 0.000,C 90.000,E1 343.196} C_DIS
LIN {X 0.091,Y -602.413,Z 1028.701,A 0.000,B 0.000,C 90.000,E1 342.127} C_DIS
LIN {X -0.358,Y -607.042,Z 1028.693,A 0.000,B 0.000,C 90.000,E1 340.859} C_DIS
LIN {X -0.199,Y -609.598,Z 1028.689,A 0.000,B 0.000,C 90.000,E1 340.061} C_DIS
LIN {X -0.276,Y -612.717,Z 1028.683,A 0.000,B 0.000,C 90.000,E1 339.028} C_DIS
LIN {X -0.121,Y -616.380,Z 1028.676,A 0.000,B 0.000,C 90.000,E1 337.720} C_DIS
LIN {X -0.155,Y -620.352,Z 1028.668,A 0.000,B 0.000,C 90.000,E1 336.177} C_DIS
LIN {X -0.177,Y -622.711,Z 1028.662,A 0.000,B 0.000,C 90.000,E1 335.153} C_DIS
LIN {X 0.134,Y -624.835,Z 1028.656,A 0.000,B 0.000,C 90.000,E1 334.101} C_DIS
LIN {X 0.190,Y -627.292,Z 1028.649,A 0.000,B 0.000,C 90.000,E1 332.820} C_DIS
LIN {X -0.315,Y -628.637,Z 1028.645,A 0.000,B 0.000,C 90.000,E1 332.103} C_DIS
LIN {X 0.098,Y -630.530,Z 1028.638,A 0.000,B 0.000,C 90.000,E1 330.795} C_DIS
LIN {X -0.005,Y -632.282,Z 1028.631,A 0.000,B 0.000,C 90.000,E1 329.537} C_DIS
LIN {X -0.083,Y -633.662,Z 1028.624,A 0.000,B 0.000,C 90.000,E1 328.280} C_DIS
LIN {X -0.346,Y -634.825,Z 1028.617,A 0.000,B 0.000,C 90.000,E1 327.041} C_DIS
LIN {X -0.056,Y -635.790,Z 1028.610,A 0.000,B 0.000,C 90.000,E1 325.754} C_DIS
LIN {X -0.305,Y -636.247,Z 1028.604,A 0.000,B 0.000,C 90.000,E1 324.769} C_DIS
LIN {X 0.345,Y -636.607,Z 1028.599,A 0.000,B 0.000,C 90.000,E1 323.703} C_DIS
LIN {X -0.134,Y -636.826,Z 1028.589,A 0.000,B 0.000,C 90.000,E1 321.984} C_DIS
LIN {X -0.328,Y -637.347,Z 1028.578,A 0.000,B 0.000,C 90.000,E1 319.989} C_DIS
LIN {X 0.421,Y -637.915,Z 1028.568,A 0.000,B 0.000,C 90.000,E1 318.162} C_DIS
LIN {X -0.104,Y -638.284,Z 1028.559,A 0.000,B 0.000,C 90.000,E1 316.701} C_DIS
LIN {X 0.168,Y -638.915,Z 1028.550,A 0.000,B 0.000,C 90.000,E1 314.919} C_DIS
LIN {X -0.072,Y -639.727,Z 1028.539,A 0.000,B 0.000,C 90.000,E1 312.933} C_DIS
LIN {X -0.040,Y -640.106,Z 1028.532,A 0.000,B 0.000,C 90.000,E1 311.676} C_DIS
LIN {X 0.054,Y -640.451,Z 1028.525,A 0.000,B 0.000,C 90.000,E1 310.415} C_DIS
LIN {X 0.069,Y -640.763,Z 1028.516,A 0.000,B 0.000,C 90.000,E1 308.910} C_DIS
LIN {X 0.172,Y -640.910,Z 1028.509,A 0.000,B 0.000,C 90.000,E1 307.649} C_DIS
LIN {X 0.221,Y -641.328,Z 1028.497,A 0.000,B 0.000,C 90.000,E1 305.391} C_DIS
LIN {X -0.076,Y -642.057,Z 1028.484,A 0.000,B 0.000,C 90.000,E1 303.166} C_DIS
LIN {X -0.132,Y -644.278,Z 1028.466,A 0.000,B 0.000,C 90.000,E1 299.922} C_DIS
LIN {X -0.324,Y -645.392,Z 1028.459,A 0.000,B 0.000,C 90.000,E1 298.693} C_DIS
LIN {X 0.384,Y -646.713,Z 1028.452,A 0.000,B 0.000,C 90.000,E1 297.385} C_DIS
LIN {X 0.060,Y -647.383,Z 1028.448,A 0.000,B 0.000,C 90.000,E1 296.668} C_DIS
LIN {X 0.126,Y -648.210,Z 1028.443,A 0.000,B 0.000,C 90.000,E1 295.668} C_DIS
LIN {X -0.192,Y -648.567,Z 1028.439,A 0.000,B 0.000,C 90.000,E1 294.951} C_DIS
LIN {X -0.195,Y -648.746,Z 1028.434,A 0.000,B 0.000,C 90.000,E1 294.207} C_DIS
LIN {X -0.101,Y -648.717,Z 1028.429,A 0.000,B 0.000,C 90.000,E1 293.206} C_DIS
LIN {X -0.171,Y -648.351,Z 1028.422,A 0.000,B 0.000,C 90.000,E1 291.972} C_DIS
LIN {X -0.011,Y -647.803,Z 1028.419,A 0.000,B 0.000,C 90.000,E1 291.461} C_DIS
LIN {X -0.093,Y -646.902,Z 1028.417,A 0.000,B 0.000,C 90.000,E1 290.972} C_DIS
LIN {X -0.251,Y -646.333,Z 1028.415,A 0.000,B 0.000,C 90.000,E1 290.737} C_DIS
LIN {X -0.147,Y -644.733,Z 1028.413,A 0.000,B 0.000,C 90.000,E1 290.355} C_DIS
LIN {X -0.306,Y -643.267,Z 1028.412,A 0.000,B 0.000,C 90.000,E1 290.120} C_DIS
LIN {X 0.328,Y -642.325,Z 1028.411,A 0.000,B 0.000,C 90.000,E1 289.939} C_DIS
LIN {X 0.353,Y -640.875,Z 1028.410,A 0.000,B 0.000,C 90.000,E1 289.812} C_DIS
LIN {X 0.102,Y -637.236,Z 1028.408,A 0.000,B 0.000,C 90.000,E1 289.450} C_DIS
LIN {X 0.120,Y -635.476,Z 1028.407,A 0.000,B 0.000,C 90.000,E1 289.322} C_DIS
LIN {X -0.097,Y -628.702,Z 1028.405,A 0.000,B 0.000,C 90.000,E1 288.960} C_DIS
LIN {X 0.344,Y -621.451,Z 1028.404,A 0.000,B 0.000,C 90.000,E1 288.598} C_DIS
LIN {X -0.100,Y -614.144,Z 1028.402,A 0.000,B 0.000,C 90.000,E1 288.362} C_DIS
LIN {X 0.074,Y -602.796,Z 1028.400,A 0.000,B 0.000,C 90.000,E1 287.946} C_DIS
LIN {X 0.035,Y -602.750,Z 1028.400,A 0.000,B 0.000,C 90.000,E1 287.946} C_DIS
LIN {X -0.179,Y -604.302,Z 1028.399,A 0.000,B 0.000,C 90.000,E1 287.764} C_DIS
LIN {X -0.227,Y -605.500,Z 1028.398,A 0.000,B 0.000,C 90.000,E1 287.638} C_DIS
LIN {X -0.005,Y -611.339,Z 1028.395,A 0.000,B 0.000,C 90.000,E1 287.094} C_DIS
LIN {X -0.145,Y -614.827,Z 1028.393,A 0.000,B 0.000,C 90.000,E1 286.732} C_DIS
LIN {X 0.201,Y -617.056,Z 1028.391,A 0.000,B 0.000,C 90.000,E1 286.441} C_DIS
LIN {X -0.064,Y -619.938,Z 1028.389,A 0.000,B 0.000,C 90.000,E1 286.079} C_DIS
LIN {X 0.279,Y -622.385,Z 1028.387,A 0.000,B 0.000,C 90.000,E1 285.662} C_DIS
LIN {X -0.154,Y -625.354,Z 1028.384,A 0.000,B 0.000,C 90.000,E1 285.190} C_DIS
LIN {X 0.039,Y -627.803,Z 1028.381,A 0.000,B 0.000,C 90.000,E1 284.662} C_DIS
LIN {X -0.206,Y -629.994,Z 1028.379,A 0.000,B 0.000,C 90.000,E1 284.175} C_DIS
LIN {X 0.209,Y -630.836,Z 1028.377,A 0.000,B 0.000,C 90.000,E1 283.883} C_DIS
LIN {X -0.175,Y -632.218,Z 1028.375,A 0.000,B 0.000,C 90.000,E1 283.411} C_DIS
LIN {X 0.066,Y -633.400,Z 1028.372,A 0.000,B 0.000,C 90.000,E1 282.883} C_DIS
LIN {X -0.118,Y -633.760,Z 1028.370,A 0.000,B 0.000,C 90.000,E1 282.647} C_DIS
LIN {X 0.135,Y -634.138,Z 1028.367,A 0.000,B 0.000,C 90.000,E1 282.119} C_DIS
LIN {X -0.358,Y -634.071,Z 1028.365,A 0.000,B 0.000,C 90.000,E1 281.658} C_DIS
LIN {X -0.099,Y -633.674,Z 1028.362,A 0.000,B 0.000,C 90.000,E1 281.130} C_DIS
LIN {X -0.282,Y -633.356,Z 1028.360,A 0.000,B 0.000,C 90.000,E1 280.894} C_DIS
LIN {X -0.032,Y -632.299,Z 1028.358,A 0.000,B 0.000,C 90.000,E1 280.366} C_DIS
LIN {X 0.099,Y -630.745,Z 1028.355,A 0.000,B 0.000,C 90.000,E1 279.849} C_DIS
LIN {X 0.327,Y -628.666,Z 1028.352,A 0.000,B 0.000,C 90.000,E1 279.321} C_DIS
LIN {X 0.026,Y -627.503,Z 1028.351,A 0.000,B 0.000,C 90.000,E1 279.095} C_DIS
LIN {X 0.227,Y -624.615,Z 1028.348,A 0.000,B 0.000,C 90.000,E1 278.568} C_DIS
LIN {X -0.149,Y -621.867,Z 1028.346,A 0.000,B 0.000,C 90.000,E1 278.219} C_DIS
LIN {X -0.305,Y -620.914,Z 1028.345,A 0.000,B 0.000,C 90.000,E1 278.106} C_DIS
LIN {X -0.241,Y -616.376,Z 1028.342,A 0.000,B 0.000,C 90.000,E1 277.587} C_DIS
LIN {X -0.192,Y -615.249,Z 1028.341,A 0.000,B 0.000,C 90.000,E1 277.466} C_DIS
LIN {X -0.253,Y -609.937,Z 1028.339,A 0.000,B 0.000,C 90.000,E1 277.004} C_DIS
LIN {X -0.284,Y -606.946,Z 1028.338,A 0.000,B 0.000,C 90.000,E1 276.777} C_DIS
LIN {X 0.021,Y -602.484,Z 1028.336,A 0.000,B 0.000,C 90.000,E1 276.429} C_DIS
LIN {X 0.272,Y -594.514,Z 1028.333,A 0.000,B 0.000,C 90.000,E1 275.910} C_DIS
LIN {X -0.244,Y -587.365,Z 1028.331,A 0.000,B 0.000,C 90.000,E1 275.625} C_DIS
LIN {X 0.085,Y -581.504,Z 1028.330,A 0.000,B 0.000,C 90.000,E1 275.391} C_DIS
LIN {X 0.071,Y -579.441,Z 1028.330,A 0.000,B 0.000,C 90.000,E1 275.334} C_DIS
LIN {X -0.062,Y -572.422,Z 1028.329,A 0.000,B 0.000,C 90.000,E1 275.220} C_DIS
LIN {X -0.104,Y -566.690,Z 1028.329,A 0.000,B 0.000,C 90.000,E1 275.163} C_DIS
LIN {X -0.147,Y -544.078,Z 1028.329,A 0.000,B 0.000,C 90.000,E1 275.163} C_DIS
LIN {X 0.266,Y -543.573,Z 1028.328,A 0.000,B 0.000,C 90.000,E1 275.049} C_DIS
LIN {X 0.179,Y -542.383,Z 1028.324,A 0.000,B 0.000,C 90.000,E1 274.245} C_DIS
LIN {X -0.018,Y -540.213,Z 1028.305,A 0.000,B 0.000,C 90.000,E1 270.859} C_DIS
LIN {X 0.061,Y -539.562,Z 1028.298,A 0.000,B 0.000,C 90.000,E1 269.714} C_DIS
LIN {X 0.141,Y -538.548,Z 1028.291,A 0.000,B 0.000,C 90.000,E1 268.282} C_DIS
LIN {X 0.250,Y -537.250,Z 1028.281,A 0.000,B 0.000,C 90.000,E1 266.560} C_DIS
LIN {X -0.162,Y -535.549,Z 1028.268,A 0.000,B 0.000,C 90.000,E1 264.318} C_DIS
LIN {X -0.051,Y -534.460,Z 1028.260,A 0.000,B 0.000,C 90.000,E1 262.875} C_DIS
LIN {X 0.036,Y -533.066,Z 1028.252,A 0.000,B 0.000,C 90.000,E1 261.432} C_DIS
LIN {X 0.085,Y -532.134,Z 1028.248,A 0.000,B 0.000,C 90.000,E1 260.566} C_DIS
LIN {X -0.049,Y -528.926,Z 1028.232,A 0.000,B 0.000,C 90.000,E1 257.701} C_DIS
LIN {X 0.219,Y -527.337,Z 1028.224,A 0.000,B 0.000,C 90.000,E1 256.228} C_DIS
LIN {X -0.054,Y -525.765,Z 1028.216,A 0.000,B 0.000,C 90.000,E1 254.810} C_DIS
LIN {X -0.060,Y -523.566,Z 1028.204,A 0.000,B 0.000,C 90.000,E1 252.779} C_DIS
LIN {X -0.106,Y -522.005,Z 1028.196,A 0.000,B 0.000,C 90.000,E1 251.329} C_DIS
LIN {X -0.034,Y -519.767,Z 1028.187,A 0.000,B 0.000,C 90.000,E1 249.571} C_DIS
LIN {X 0.159,Y -517.443,Z 1028.177,A 0.000,B 0.000,C 90.000,E1 247.794} C_DIS
LIN {X -0.116,Y -515.514,Z 1028.169,A 0.000,B 0.000,C 90.000,E1 246.357} C_DIS
LIN {X -0.080,Y -513.858,Z 1028.162,A 0.000,B 0.000,C 90.000,E1 245.177} C_DIS
LIN {X 0.140,Y -512.032,Z 1028.156,A 0.000,B 0.000,C 90.000,E1 243.973} C_DIS
LIN {X 0.203,Y -509.641,Z 1028.147,A 0.000,B 0.000,C 90.000,E1 242.487} C_DIS
LIN {X -0.222,Y -507.111,Z 1028.139,A 0.000,B 0.000,C 90.000,E1 241.051} C_DIS
LIN {X -0.122,Y -503.913,Z 1028.129,A 0.000,B 0.000,C 90.000,E1 239.253} C_DIS
LIN {X 0.028,Y -501.136,Z 1028.121,A 0.000,B 0.000,C 90.000,E1 237.740} C_DIS
LIN {X -0.057,Y -498.731,Z 1028.114,A 0.000,B 0.000,C 90.000,E1 236.548} C_DIS
LIN {X -0.036,Y -496.185,Z 1028.107,A 0.000,B 0.000,C 90.000,E1 235.341} C_DIS
LIN {X 0.240,Y -494.122,Z 1028.102,A 0.000,B 0.000,C 90.000,E1 234.402} C_DIS
LIN {X -0.093,Y -490.605,Z 1028.094,A 0.000,B 0.000,C 90.000,E1 232.924} C_DIS
LIN {X 0.103,Y -486.970,Z 1028.086,A 0.000,B 0.000,C 90.000,E1 231.376} C_DIS
LIN {X -0.009,Y -481.412,Z 1028.072,A 0.000,B 0.000,C 90.000,E1 228.933} C_DIS
LIN {X -0.025,Y -476.000,Z 1028.058,A 0.000,B 0.000,C 90.000,E1 226.458} C_DIS
LIN {X -0.078,Y -472.148,Z 1028.048,A 0.000,B 0.000,C 90.000,E1 224.595} C_DIS
LIN {X 0.196,Y -467.615,Z 1028.036,A 0.000,B 0.000,C 90.000,E1 222.366} C_DIS
LIN {X -0.096,Y -464.421,Z 1028.027,A 0.000,B 0.000,C 90.000,E1 220.825} C_DIS
LIN {X 0.256,Y -461.148,Z 1028.018,A 0.000,B 0.000,C 90.000,E1 219.197} C_DIS
LIN {X -0.122,Y -458.237,Z 1028.011,A 0.000,B 0.000,C 90.000,E1 217.971} C_DIS
LIN {X 0.192,Y -453.947,Z 1028.000,A 0.000,B 0.000,C 90.000,E1 216.011} C_DIS
LIN {X 0.153,Y -450.520,Z 1027.991,A 0.000,B 0.000,C 90.000,E1 214.405} C_DIS
LIN {X 0.045,Y -447.066,Z 1027.982,A 0.000,B 0.000,C 90.000,E1 212.801} C_DIS
LIN {X -0.174,Y -442.814,Z 1027.971,A 0.000,B 0.000,C 90.000,E1 210.875} C_DIS
LIN {X 0.034,Y -439.951,Z 1027.964,A 0.000,B 0.000,C 90.000,E1 209.539} C_DIS
LIN {X 0.007,Y -436.184,Z 1027.955,A 0.000,B 0.000,C 90.000,E1 207.897} C_DIS
LIN {X -0.099,Y -431.640,Z 1027.944,A 0.000,B 0.000,C 90.000,E1 205.924} C_DIS
LIN {X 0.057,Y -426.469,Z 1027.931,A 0.000,B 0.000,C 90.000,E1 203.567} C_DIS
LIN {X -0.053,Y -421.597,Z 1027.918,A 0.000,B 0.000,C 90.000,E1 201.227} C_DIS
LIN {X -0.116,Y -415.993,Z 1027.901,A 0.000,B 0.000,C 90.000,E1 198.181} C_DIS
LIN {X -0.080,Y -409.952,Z 1027.878,A 0.000,B 0.000,C 90.000,E1 194.064} C_DIS
LIN {X -0.191,Y -407.959,Z 1027.869,A 0.000,B 0.000,C 90.000,E1 192.355} C_DIS
LIN {X -0.157,Y -407.425,Z 1027.865,A 0.000,B 0.000,C 90.000,E1 191.658} C_DIS
LIN {X -0.045,Y -407.106,Z 1027.861,A 0.000,B 0.000,C 90.000,E1 190.950} C_DIS
LIN {X 0.065,Y -407.255,Z 1027.857,A 0.000,B 0.000,C 90.000,E1 190.254} C_DIS
LIN {X 0.123,Y -407.850,Z 1027.854,A 0.000,B 0.000,C 90.000,E1 189.726} C_DIS
LIN {X 0.097,Y -408.109,Z 1027.853,A 0.000,B 0.000,C 90.000,E1 189.557} C_DIS
LIN {X 0.105,Y -409.787,Z 1027.850,A 0.000,B 0.000,C 90.000,E1 188.973} C_DIS
LIN {X 0.111,Y -411.884,Z 1027.847,A 0.000,B 0.000,C 90.000,E1 188.454} C_DIS
LIN {X 0.156,Y -413.663,Z 1027.845,A 0.000,B 0.000,C 90.000,E1 188.106} C_DIS
LIN {X 0.015,Y -417.670,Z 1027.842,A 0.000,B 0.000,C 90.000,E1 187.466} C_DIS
LIN {X -0.010,Y -426.021,Z 1027.835,A 0.000,B 0.000,C 90.000,E1 186.315} C_DIS
LIN {X 0.080,Y -436.161,Z 1027.828,A 0.000,B 0.000,C 90.000,E1 184.992} C_DIS
LIN {X 0.100,Y -444.646,Z 1027.822,A 0.000,B 0.000,C 90.000,E1 183.898} C_DIS
LIN {X 0.013,Y -450.980,Z 1027.817,A 0.000,B 0.000,C 90.000,E1 183.094} C_DIS
LIN {X 0.213,Y -457.032,Z 1027.813,A 0.000,B 0.000,C 90.000,E1 182.293} C_DIS
LIN {X 0.084,Y -465.611,Z 1027.807,A 0.000,B 0.000,C 90.000,E1 181.203} C_DIS
LIN {X 0.203,Y -474.733,Z 1027.800,A 0.000,B 0.000,C 90.000,E1 179.943} C_DIS
LIN {X 0.062,Y -481.280,Z 1027.795,A 0.000,B 0.000,C 90.000,E1 179.026} C_DIS
LIN {X 0.003,Y -487.746,Z 1027.790,A 0.000,B 0.000,C 90.000,E1 178.108} C_DIS
LIN {X 0.001,Y -494.028,Z 1027.784,A 0.000,B 0.000,C 90.000,E1 177.192} C_DIS
LIN {X -0.227,Y -500.899,Z 1027.779,A 0.000,B 0.000,C 90.000,E1 176.159} C_DIS
LIN {X 0.174,Y -507.585,Z 1027.773,A 0.000,B 0.000,C 90.000,E1 175.065} C_DIS
LIN {X 0.116,Y -515.639,Z 1027.765,A 0.000,B 0.000,C 90.000,E1 173.742} C_DIS
LIN {X -0.081,Y -525.830,Z 1027.756,A 0.000,B 0.000,C 90.000,E1 172.008} C_DIS
LIN {X 0.190,Y -529.990,Z 1027.752,A 0.000,B 0.000,C 90.000,E1 171.254} C_DIS
LIN {X 0.270,Y -536.525,Z 1027.745,A 0.000,B 0.000,C 90.000,E1 170.095} C_DIS
LIN {X -0.015,Y -544.719,Z 1027.737,A 0.000,B 0.000,C 90.000,E1 168.701} C_DIS
LIN {X -0.059,Y -552.620,Z 1027.729,A 0.000,B 0.000,C 90.000,E1 167.297} C_DIS
LIN {X 0.033,Y -556.362,Z 1027.726,A 0.000,B 0.000,C 90.000,E1 166.589} C_DIS
LIN {X 0.176,Y -562.268,Z 1027.719,A 0.000,B 0.000,C 90.000,E1 165.463} C_DIS
LIN {X -0.139,Y -568.138,Z 1027.713,A 0.000,B 0.000,C 90.000,E1 164.393} C_DIS
LIN {X -0.027,Y -575.156,Z 1027.706,A 0.000,B 0.000,C 90.000,E1 163.015} C_DIS
LIN {X 0.177,Y -579.092,Z 1027.701,A 0.000,B 0.000,C 90.000,E1 162.181} C_DIS
LIN {X -0.216,Y -583.481,Z 1027.696,A 0.000,B 0.000,C 90.000,E1 161.275} C_DIS
LIN {X -0.082,Y -588.064,Z 1027.690,A 0.000,B 0.000,C 90.000,E1 160.188} C_DIS
LIN {X 0.317,Y -592.505,Z 1027.684,A 0.000,B 0.000,C 90.000,E1 159.082} C_DIS
LIN {X 0.008,Y -596.705,Z 1027.678,A 0.000,B 0.000,C 90.000,E1 158.050} C_DIS
LIN {X 0.206,Y -600.535,Z 1027.672,A 0.000,B 0.000,C 90.000,E1 156.975} C_DIS
LIN {X -0.256,Y -603.268,Z 1027.668,A 0.000,B 0.000,C 90.000,E1 156.230} C_DIS
LIN {X -0.262,Y -607.444,Z 1027.661,A 0.000,B 0.000,C 90.000,E1 154.921} C_DIS
LIN {X 0.053,Y -611.327,Z 1027.653,A 0.000,B 0.000,C 90.000,E1 153.589} C_DIS
LIN {X -0.056,Y -613.541,Z 1027.649,A 0.000,B 0.000,C 90.000,E1 152.820} C_DIS
LIN {X 0.077,Y -617.589,Z 1027.640,A 0.000,B 0.000,C 90.000,E1 151.257} C_DIS
LIN {X -0.224,Y -620.180,Z 1027.635,A 0.000,B 0.000,C 90.000,E1 150.255} C_DIS
LIN {X 0.045,Y -623.500,Z 1027.628,A 0.000,B 0.000,C 90.000,E1 148.948} C_DIS
LIN {X -0.378,Y -627.260,Z 1027.619,A 0.000,B 0.000,C 90.000,E1 147.454} C_DIS
LIN {X 0.140,Y -630.345,Z 1027.612,A 0.000,B 0.000,C 90.000,E1 146.135} C_DIS
LIN {X 0.212,Y -634.043,Z 1027.604,A 0.000,B 0.000,C 90.000,E1 144.609} C_DIS
LIN {X -0.169,Y -637.653,Z 1027.595,A 0.000,B 0.000,C 90.000,E1 143.130} C_DIS
LIN {X -0.104,Y -641.260,Z 1027.587,A 0.000,B 0.000,C 90.000,E1 141.618} C_DIS
LIN {X 0.020,Y -644.252,Z 1027.580,A 0.000,B 0.000,C 90.000,E1 140.356} C_DIS
LIN {X 0.122,Y -647.768,Z 1027.572,A 0.000,B 0.000,C 90.000,E1 138.852} C_DIS
LIN {X 0.083,Y -653.816,Z 1027.558,A 0.000,B 0.000,C 90.000,E1 136.377} C_DIS
LIN {X -0.251,Y -660.512,Z 1027.544,A 0.000,B 0.000,C 90.000,E1 133.947} C_DIS
LIN {X 0.130,Y -664.876,Z 1027.536,A 0.000,B 0.000,C 90.000,E1 132.447} C_DIS
LIN {X 0.152,Y -667.784,Z 1027.531,A 0.000,B 0.000,C 90.000,E1 131.472} C_DIS
LIN {X -0.290,Y -670.653,Z 1027.525,A 0.000,B 0.000,C 90.000,E1 130.539} C_DIS
LIN {X -0.191,Y -673.391,Z 1027.520,A 0.000,B 0.000,C 90.000,E1 129.564} C_DIS
LIN {X 0.059,Y -676.748,Z 1027.513,A 0.000,B 0.000,C 90.000,E1 128.338} C_DIS
LIN {X 0.391,Y -680.583,Z 1027.505,A 0.000,B 0.000,C 90.000,E1 126.870} C_DIS
LIN {X -0.004,Y -685.012,Z 1027.496,A 0.000,B 0.000,C 90.000,E1 125.231} C_DIS
LIN {X 0.030,Y -688.088,Z 1027.489,A 0.000,B 0.000,C 90.000,E1 124.040} C_DIS
LIN {X -0.274,Y -691.058,Z 1027.483,A 0.000,B 0.000,C 90.000,E1 122.880} C_DIS
LIN {X 0.057,Y -693.989,Z 1027.476,A 0.000,B 0.000,C 90.000,E1 121.671} C_DIS
LIN {X 0.191,Y -696.167,Z 1027.471,A 0.000,B 0.000,C 90.000,E1 120.718} C_DIS
LIN {X -0.007,Y -698.026,Z 1027.466,A 0.000,B 0.000,C 90.000,E1 119.795} C_DIS
LIN {X -0.182,Y -699.542,Z 1027.460,A 0.000,B 0.000,C 90.000,E1 118.871} C_DIS
LIN {X 0.275,Y -700.769,Z 1027.455,A 0.000,B 0.000,C 90.000,E1 117.897} C_DIS
LIN {X -0.198,Y -701.680,Z 1027.450,A 0.000,B 0.000,C 90.000,E1 117.001} C_DIS
LIN {X 0.255,Y -702.753,Z 1027.443,A 0.000,B 0.000,C 90.000,E1 115.796} C_DIS
LIN {X -0.191,Y -703.463,Z 1027.438,A 0.000,B 0.000,C 90.000,E1 114.899} C_DIS
LIN {X 0.372,Y -703.554,Z 1027.436,A 0.000,B 0.000,C 90.000,E1 114.387} C_DIS
LIN {X -0.277,Y -703.530,Z 1027.434,A 0.000,B 0.000,C 90.000,E1 114.207} C_DIS
LIN {X 0.283,Y -702.821,Z 1027.432,A 0.000,B 0.000,C 90.000,E1 113.695} C_DIS
LIN {X -0.364,Y -702.322,Z 1027.431,A 0.000,B 0.000,C 90.000,E1 113.515} C_DIS
LIN {X 0.048,Y -700.579,Z 1027.429,A 0.000,B 0.000,C 90.000,E1 113.131} C_DIS
LIN {X 0.044,Y -699.270,Z 1027.427,A 0.000,B 0.000,C 90.000,E1 112.898} C_DIS
LIN {X 0.177,Y -698.504,Z 1027.427,A 0.000,B 0.000,C 90.000,E1 112.770} C_DIS
LIN {X 0.307,Y -697.371,Z 1027.426,A 0.000,B 0.000,C 90.000,E1 112.642} C_DIS
LIN {X 0.436,Y -695.657,Z 1027.425,A 0.000,B 0.000,C 90.000,E1 112.514} C_DIS
LIN {X 0.305,Y -689.329,Z 1027.423,A 0.000,B 0.000,C 90.000,E1 112.153} C_DIS
LIN {X 0.175,Y -686.963,Z 1027.423,A 0.000,B 0.000,C 90.000,E1 112.078} C_DIS
LIN {X -0.213,Y -684.145,Z 1027.422,A 0.000,B 0.000,C 90.000,E1 112.025} C_DIS
LIN {X -0.011,Y -675.737,Z 1027.422,A 0.000,B 0.000,C 90.000,E1 111.897} C_DIS
LIN {X -0.073,Y -613.371,Z 1027.422,A 0.000,B 0.000,C 90.000,E1 111.897} C_DIS
LIN {X 0.106,Y -611.773,Z 1027.422,A 0.000,B 0.000,C 90.000,E1 111.844} C_DIS
LIN {X -0.116,Y -605.173,Z 1027.420,A 0.000,B 0.000,C 90.000,E1 111.642} C_DIS
LIN {X -0.042,Y -598.695,Z 1027.419,A 0.000,B 0.000,C 90.000,E1 111.334} C_DIS
LIN {X 0.167,Y -593.128,Z 1027.417,A 0.000,B 0.000,C 90.000,E1 110.972} C_DIS
LIN {X 0.358,Y -586.874,Z 1027.414,A 0.000,B 0.000,C 90.000,E1 110.482} C_DIS
LIN {X -0.012,Y -577.371,Z 1027.410,A 0.000,B 0.000,C 90.000,E1 109.704} C_DIS
LIN {X -0.232,Y -571.182,Z 1027.407,A 0.000,B 0.000,C 90.000,E1 109.268} C_DIS
LIN {X -0.002,Y -569.606,Z 1027.406,A 0.000,B 0.000,C 90.000,E1 109.141} C_DIS
LIN {X 0.016,Y -561.288,Z 1027.404,A 0.000,B 0.000,C 90.000,E1 108.671} C_DIS
LIN {X -0.301,Y -554.701,Z 1027.402,A 0.000,B 0.000,C 90.000,E1 108.362} C_DIS
LIN {X 0.090,Y -549.595,Z 1027.400,A 0.000,B 0.000,C 90.000,E1 108.000} C_DIS
LIN {X 0.154,Y -548.129,Z 1027.399,A 0.000,B 0.000,C 90.000,E1 107.819} C_DIS
LIN {X 0.112,Y -548.115,Z 1027.399,A 0.000,B 0.000,C 90.000,E1 107.819} C_DIS
LIN {X 0.283,Y -547.759,Z 1027.397,A 0.000,B 0.000,C 90.000,E1 107.511} C_DIS
LIN {X 0.142,Y -548.825,Z 1027.384,A 0.000,B 0.000,C 90.000,E1 105.134} C_DIS
LIN {X -0.026,Y -550.787,Z 1027.367,A 0.000,B 0.000,C 90.000,E1 102.063} C_DIS
LIN {X -0.043,Y -553.570,Z 1027.351,A 0.000,B 0.000,C 90.000,E1 99.265} C_DIS
LIN {X -0.066,Y -555.185,Z 1027.344,A 0.000,B 0.000,C 90.000,E1 97.871} C_DIS
LIN {X -0.141,Y -556.751,Z 1027.336,A 0.000,B 0.000,C 90.000,E1 96.486} C_DIS
LIN {X -0.248,Y -558.115,Z 1027.328,A 0.000,B 0.000,C 90.000,E1 95.106} C_DIS
LIN {X 0.029,Y -558.760,Z 1027.324,A 0.000,B 0.000,C 90.000,E1 94.245} C_DIS
LIN {X -0.039,Y -559.609,Z 1027.316,A 0.000,B 0.000,C 90.000,E1 92.865} C_DIS
LIN {X -0.222,Y -560.154,Z 1027.310,A 0.000,B 0.000,C 90.000,E1 91.776} C_DIS
LIN {X -0.223,Y -560.816,Z 1027.301,A 0.000,B 0.000,C 90.000,E1 90.115} C_DIS
LIN {X -0.095,Y -561.492,Z 1027.290,A 0.000,B 0.000,C 90.000,E1 88.165} C_DIS
LIN {X -0.143,Y -561.938,Z 1027.282,A 0.000,B 0.000,C 90.000,E1 86.788} C_DIS
LIN {X -0.055,Y -562.327,Z 1027.273,A 0.000,B 0.000,C 90.000,E1 85.122} C_DIS
LIN {X -0.059,Y -562.670,Z 1027.265,A 0.000,B 0.000,C 90.000,E1 83.742} C_DIS
LIN {X -0.012,Y -563.277,Z 1027.251,A 0.000,B 0.000,C 90.000,E1 81.254} C_DIS
LIN {X -0.187,Y -563.903,Z 1027.241,A 0.000,B 0.000,C 90.000,E1 79.342} C_DIS
LIN {X 0.021,Y -564.943,Z 1027.229,A 0.000,B 0.000,C 90.000,E1 77.117} C_DIS
LIN {X 0.216,Y -566.129,Z 1027.218,A 0.000,B 0.000,C 90.000,E1 75.172} C_DIS
LIN {X -0.180,Y -567.782,Z 1027.206,A 0.000,B 0.000,C 90.000,E1 73.015} C_DIS
LIN {X 0.050,Y -569.059,Z 1027.196,A 0.000,B 0.000,C 90.000,E1 71.348} C_DIS
LIN {X -0.062,Y -570.486,Z 1027.186,A 0.000,B 0.000,C 90.000,E1 69.444} C_DIS
LIN {X -0.126,Y -571.765,Z 1027.175,A 0.000,B 0.000,C 90.000,E1 67.539} C_DIS
LIN {X -0.310,Y -572.678,Z 1027.166,A 0.000,B 0.000,C 90.000,E1 65.921} C_DIS
LIN {X -0.246,Y -573.474,Z 1027.157,A 0.000,B 0.000,C 90.000,E1 64.280} C_DIS
LIN {X 0.084,Y -574.181,Z 1027.148,A 0.000,B 0.000,C 90.000,E1 62.615} C_DIS
LIN {X 0.072,Y -574.739,Z 1027.140,A 0.000,B 0.000,C 90.000,E1 61.257} C_DIS
LIN {X -0.153,Y -575.215,Z 1027.133,A 0.000,B 0.000,C 90.000,E1 59.921} C_DIS
LIN {X 0.130,Y -575.644,Z 1027.125,A 0.000,B 0.000,C 90.000,E1 58.535} C_DIS
LIN {X 0.210,Y -576.256,Z 1027.115,A 0.000,B 0.000,C 90.000,E1 56.628} C_DIS
LIN {X -0.004,Y -576.490,Z 1027.106,A 0.000,B 0.000,C 90.000,E1 55.022} C_DIS
LIN {X 0.281,Y -576.495,Z 1027.100,A 0.000,B 0.000,C 90.000,E1 53.909} C_DIS
LIN {X -0.054,Y -576.331,Z 1027.091,A 0.000,B 0.000,C 90.000,E1 52.316} C_DIS
LIN {X -0.249,Y -575.958,Z 1027.085,A 0.000,B 0.000,C 90.000,E1 51.251} C_DIS
LIN {X -0.247,Y -575.145,Z 1027.076,A 0.000,B 0.000,C 90.000,E1 49.622} C_DIS
LIN {X -0.031,Y -574.210,Z 1027.068,A 0.000,B 0.000,C 90.000,E1 48.243} C_DIS
LIN {X 0.038,Y -573.239,Z 1027.062,A 0.000,B 0.000,C 90.000,E1 47.148} C_DIS
LIN {X -0.026,Y -572.381,Z 1027.057,A 0.000,B 0.000,C 90.000,E1 46.338} C_DIS
LIN {X -0.200,Y -571.764,Z 1027.054,A 0.000,B 0.000,C 90.000,E1 45.810} C_DIS
LIN {X -0.279,Y -570.567,Z 1027.050,A 0.000,B 0.000,C 90.000,E1 45.000} C_DIS
LIN {X 0.133,Y -568.698,Z 1027.044,A 0.000,B 0.000,C 90.000,E1 43.866} C_DIS
LIN {X 0.122,Y -566.624,Z 1027.038,A 0.000,B 0.000,C 90.000,E1 42.771} C_DIS
LIN {X -0.021,Y -564.805,Z 1027.033,A 0.000,B 0.000,C 90.000,E1 41.962} C_DIS
LIN {X 0.182,Y -563.508,Z 1027.030,A 0.000,B 0.000,C 90.000,E1 41.391} C_DIS
LIN {X -0.370,Y -561.229,Z 1027.026,A 0.000,B 0.000,C 90.000,E1 40.620} C_DIS
LIN {X 0.181,Y -559.644,Z 1027.022,A 0.000,B 0.000,C 90.000,E1 40.011} C_DIS
LIN {X 0.015,Y -556.879,Z 1027.018,A 0.000,B 0.000,C 90.000,E1 39.197} C_DIS
LIN {X -0.179,Y -553.874,Z 1027.013,A 0.000,B 0.000,C 90.000,E1 38.382} C_DIS
LIN {X -0.037,Y -551.719,Z 1027.010,A 0.000,B 0.000,C 90.000,E1 37.810} C_DIS
LIN {X 0.151,Y -548.156,Z 1027.005,A 0.000,B 0.000,C 90.000,E1 36.950} C_DIS
LIN {X 0.293,Y -544.322,Z 1027.001,A 0.000,B 0.000,C 90.000,E1 36.091} C_DIS
LIN {X 0.097,Y -538.765,Z 1026.994,A 0.000,B 0.000,C 90.000,E1 34.978} C_DIS
LIN {X 0.128,Y -534.235,Z 1026.990,A 0.000,B 0.000,C 90.000,E1 34.119} C_DIS
LIN {X -0.180,Y -531.066,Z 1026.986,A 0.000,B 0.000,C 90.000,E1 33.579} C_DIS
LIN {X 0.198,Y -526.059,Z 1026.982,A 0.000,B 0.000,C 90.000,E1 32.673} C_DIS
LIN {X 0.118,Y -521.548,Z 1026.978,A 0.000,B 0.000,C 90.000,E1 31.957} C_DIS
LIN {X 0.002,Y -517.689,Z 1026.974,A 0.000,B 0.000,C 90.000,E1 31.386} C_DIS
LIN {X 0.030,Y -513.541,Z 1026.971,A 0.000,B 0.000,C 90.000,E1 30.797} C_DIS
LIN {X 0.207,Y -510.306,Z 1026.969,A 0.000,B 0.000,C 90.000,E1 30.335} C_DIS
LIN {X 0.109,Y -504.491,Z 1026.965,A 0.000,B 0.000,C 90.000,E1 29.617} C_DIS
LIN {X -0.203,Y -500.708,Z 1026.962,A 0.000,B 0.000,C 90.000,E1 29.205} C_DIS
LIN {X 0.196,Y -495.490,Z 1026.959,A 0.000,B 0.000,C 90.000,E1 28.565} C_DIS
LIN {X -0.012,Y -491.432,Z 1026.956,A 0.000,B 0.000,C 90.000,E1 28.153} C_DIS
LIN {X -0.053,Y -481.807,Z 1026.951,A 0.000,B 0.000,C 90.000,E1 27.180} C_DIS
LIN {X -0.144,Y -473.085,Z 1026.946,A 0.000,B 0.000,C 90.000,E1 26.360} C_DIS
LIN {X -0.161,Y -461.331,Z 1026.940,A 0.000,B 0.000,C 90.000,E1 25.283} C_DIS
LIN {X 0.181,Y -449.192,Z 1026.935,A 0.000,B 0.000,C 90.000,E1 24.207} C_DIS
LIN {X -0.180,Y -434.077,Z 1026.927,A 0.000,B 0.000,C 90.000,E1 22.950} C_DIS
LIN {X 0.070,Y -416.501,Z 1026.918,A 0.000,B 0.000,C 90.000,E1 21.227} C_DIS
LIN {X 0.004,Y -402.387,Z 1026.910,A 0.000,B 0.000,C 90.000,E1 19.704} C_DIS
LIN {X -0.070,Y -398.416,Z 1026.907,A 0.000,B 0.000,C 90.000,E1 19.214} C_DIS
LIN {X -0.021,Y -397.208,Z 1026.906,A 0.000,B 0.000,C 90.000,E1 19.033} C_DIS
LIN {X 0.233,Y -394.757,Z 1026.904,A 0.000,B 0.000,C 90.000,E1 18.598} C_DIS
LIN {X -0.106,Y -393.603,Z 1026.903,A 0.000,B 0.000,C 90.000,E1 18.471} C_DIS
LIN {X -0.075,Y -392.800,Z 1026.902,A 0.000,B 0.000,C 90.000,E1 18.290} C_DIS
LIN {X -0.046,Y -392.173,Z 1026.901,A 0.000,B 0.000,C 90.000,E1 18.109} C_DIS
LIN {X 0.123,Y -391.335,Z 1026.897,A 0.000,B 0.000,C 90.000,E1 17.457} C_DIS
LIN {X 0.147,Y -391.166,Z 1026.896,A 0.000,B 0.000,C 90.000,E1 17.275} C_DIS
LIN {X 0.215,Y -391.220,Z 1026.893,A 0.000,B 0.000,C 90.000,E1 16.732} C_DIS
LIN {X -0.127,Y -391.975,Z 1026.887,A 0.000,B 0.000,C 90.000,E1 15.717} C_DIS
LIN {X -0.183,Y -395.607,Z 1026.870,A 0.000,B 0.000,C 90.000,E1 12.535} C_DIS
LIN {X 0.025,Y -402.695,Z 1026.844,A 0.000,B 0.000,C 90.000,E1 7.936} C_DIS
LIN {X -0.078,Y -408.997,Z 1026.827,A 0.000,B 0.000,C 90.000,E1 4.821} C_DIS
LIN {X -0.064,Y -413.659,Z 1026.815,A 0.000,B 0.000,C 90.000,E1 2.751} C_DIS
LIN {X -0.062,Y -414.684,Z 1026.813,A 0.000,B 0.000,C 90.000,E1 2.407} C_DIS
LIN {X -0.170,Y -416.519,Z 1026.811,A 0.000,B 0.000,C 90.000,E1 1.949} C_DIS
LIN {X -0.151,Y -417.514,Z 1026.810,A 0.000,B 0.000,C 90.000,E1 1.776} C_DIS
LIN {X 0.034,Y -422.989,Z 1026.806,A 0.000,B 0.000,C 90.000,E1 1.088} C_DIS
LIN {X 0.134,Y -427.468,Z 1026.804,A 0.000,B 0.000,C 90.000,E1 0.745} C_DIS
LIN {X -0.004,Y -434.750,Z 1026.802,A 0.000,B 0.000,C 90.000,E1 0.344} C_DIS
LIN {X 0.023,Y -455.388,Z 1026.795,A 0.000,B 0.000,C 90.000,E1 359.083} C_DIS
LIN {X 0.102,Y -468.637,Z 1026.791,A 0.000,B 0.000,C 90.000,E1 358.282} C_DIS
LIN {X 0.221,Y -481.805,Z 1026.786,A 0.000,B 0.000,C 90.000,E1 357.478} C_DIS
LIN {X -0.193,Y -493.232,Z 1026.782,A 0.000,B 0.000,C 90.000,E1 356.846} C_DIS
LIN {X 0.004,Y -502.837,Z 1026.779,A 0.000,B 0.000,C 90.000,E1 356.216} C_DIS
LIN {X 0.005,Y -510.730,Z 1026.776,A 0.000,B 0.000,C 90.000,E1 355.698} C_DIS
LIN {X -0.206,Y -518.295,Z 1026.773,A 0.000,B 0.000,C 90.000,E1 355.179} C_DIS
LIN {X -0.243,Y -524.296,Z 1026.771,A 0.000,B 0.000,C 90.000,E1 354.723} C_DIS
LIN {X 0.193,Y -531.288,Z 1026.767,A 0.000,B 0.000,C 90.000,E1 354.090} C_DIS
LIN {X -0.166,Y -536.916,Z 1026.765,A 0.000,B 0.000,C 90.000,E1 353.628} C_DIS
LIN {X 0.029,Y -540.995,Z 1026.762,A 0.000,B 0.000,C 90.000,E1 353.223} C_DIS
LIN {X -0.030,Y -547.178,Z 1026.759,A 0.000,B 0.000,C 90.000,E1 352.591} C_DIS
LIN {X -0.053,Y -553.121,Z 1026.755,A 0.000,B 0.000,C 90.000,E1 351.894} C_DIS
LIN {X 0.186,Y -557.523,Z 1026.752,A 0.000,B 0.000,C 90.000,E1 351.319} C_DIS
LIN {X 0.214,Y -562.372,Z 1026.748,A 0.000,B 0.000,C 90.000,E1 350.622} C_DIS
LIN {X -0.030,Y -566.008,Z 1026.745,A 0.000,B 0.000,C 90.000,E1 350.095} C_DIS
LIN {X 0.017,Y -572.522,Z 1026.739,A 0.000,B 0.000,C 90.000,E1 348.993} C_DIS
LIN {X 0.288,Y -576.190,Z 1026.735,A 0.000,B 0.000,C 90.000,E1 348.285} C_DIS
LIN {X -0.088,Y -579.528,Z 1026.731,A 0.000,B 0.000,C 90.000,E1 347.645} C_DIS
LIN {X 0.155,Y -585.132,Z 1026.725,A 0.000,B 0.000,C 90.000,E1 346.408} C_DIS
LIN {X 0.146,Y -589.772,Z 1026.719,A 0.000,B 0.000,C 90.000,E1 345.338} C_DIS
LIN {X 0.043,Y -594.185,Z 1026.713,A 0.000,B 0.000,C 90.000,E1 344.283} C_DIS
LIN {X 0.321,Y -598.449,Z 1026.707,A 0.000,B 0.000,C 90.000,E1 343.196} C_DIS
LIN {X -0.084,Y -602.460,Z 1026.701,A 0.000,B 0.000,C 90.000,E1 342.181} C_DIS
LIN {X 0.044,Y -607.139,Z 1026.694,A 0.000,B 0.000,C 90.000,E1 340.859} C_DIS
LIN {X 0.206,Y -609.737,Z 1026.689,A 0.000,B 0.000,C 90.000,E1 340.061} C_DIS
LIN {X 0.088,Y -613.640,Z 1026.682,A 0.000,B 0.000,C 90.000,E1 338.773} C_DIS
LIN {X 0.031,Y -617.253,Z 1026.675,A 0.000,B 0.000,C 90.000,E1 337.486} C_DIS
LIN {X 0.257,Y -621.248,Z 1026.666,A 0.000,B 0.000,C 90.000,E1 335.921} C_DIS
LIN {X -0.013,Y -623.552,Z 1026.661,A 0.000,B 0.000,C 90.000,E1 334.921} C_DIS
LIN {X 0.013,Y -625.642,Z 1026.655,A 0.000,B 0.000,C 90.000,E1 333.896} C_DIS
LIN {X 0.087,Y -628.125,Z 1026.648,A 0.000,B 0.000,C 90.000,E1 332.615} C_DIS
LIN {X 0.149,Y -629.405,Z 1026.644,A 0.000,B 0.000,C 90.000,E1 331.847} C_DIS
LIN {X 0.025,Y -631.286,Z 1026.637,A 0.000,B 0.000,C 90.000,E1 330.589} C_DIS
LIN {X -0.092,Y -632.714,Z 1026.631,A 0.000,B 0.000,C 90.000,E1 329.587} C_DIS
LIN {X -0.156,Y -634.140,Z 1026.624,A 0.000,B 0.000,C 90.000,E1 328.329} C_DIS
LIN {X 0.157,Y -635.562,Z 1026.616,A 0.000,B 0.000,C 90.000,E1 326.786} C_DIS
LIN {X -0.075,Y -636.507,Z 1026.609,A 0.000,B 0.000,C 90.000,E1 325.548} C_DIS
LIN {X 0.056,Y -636.958,Z 1026.603,A 0.000,B 0.000,C 90.000,E1 324.529} C_DIS
LIN {X -0.168,Y -637.278,Z 1026.597,A 0.000,B 0.000,C 90.000,E1 323.543} C_DIS
LIN {X -0.005,Y -637.499,Z 1026.590,A 0.000,B 0.000,C 90.000,E1 322.271} C_DIS
LIN {X -0.178,Y -637.960,Z 1026.579,A 0.000,B 0.000,C 90.000,E1 320.275} C_DIS
LIN {X 0.073,Y -638.665,Z 1026.568,A 0.000,B 0.000,C 90.000,E1 318.243} C_DIS
LIN {X 0.000,Y -639.065,Z 1026.560,A 0.000,B 0.000,C 90.000,E1 316.743} C_DIS
LIN {X -0.235,Y -639.824,Z 1026.549,A 0.000,B 0.000,C 90.000,E1 314.757} C_DIS
LIN {X 0.071,Y -640.550,Z 1026.539,A 0.000,B 0.000,C 90.000,E1 312.975} C_DIS
LIN {X -0.148,Y -640.872,Z 1026.535,A 0.000,B 0.000,C 90.000,E1 312.243} C_DIS
LIN {X 0.297,Y -641.336,Z 1026.526,A 0.000,B 0.000,C 90.000,E1 310.701} C_DIS
LIN {X -0.078,Y -641.622,Z 1026.519,A 0.000,B 0.000,C 90.000,E1 309.483} C_DIS
LIN {X 0.049,Y -641.969,Z 1026.511,A 0.000,B 0.000,C 90.000,E1 307.971} C_DIS
LIN {X 0.083,Y -642.159,Z 1026.501,A 0.000,B 0.000,C 90.000,E1 306.217} C_DIS
LIN {X -0.042,Y -642.499,Z 1026.494,A 0.000,B 0.000,C 90.000,E1 304.978} C_DIS
LIN {X -0.303,Y -643.295,Z 1026.482,A 0.000,B 0.000,C 90.000,E1 302.752} C_DIS
LIN {X -0.226,Y -645.272,Z 1026.467,A 0.000,B 0.000,C 90.000,E1 300.001} C_DIS
LIN {X 0.248,Y -647.502,Z 1026.454,A 0.000,B 0.000,C 90.000,E1 297.719} C_DIS
LIN {X 0.027,Y -648.497,Z 1026.449,A 0.000,B 0.000,C 90.000,E1 296.744} C_DIS
LIN {X -0.100,Y -649.560,Z 1026.442,A 0.000,B 0.000,C 90.000,E1 295.515} C_DIS
LIN {X -0.004,Y -649.998,Z 1026.436,A 0.000,B 0.000,C 90.000,E1 294.515} C_DIS
LIN {X 0.012,Y -650.119,Z 1026.432,A 0.000,B 0.000,C 90.000,E1 293.770} C_DIS
LIN {X 0.214,Y -649.942,Z 1026.425,A 0.000,B 0.000,C 90.000,E1 292.514} C_DIS
LIN {X 0.143,Y -649.795,Z 1026.422,A 0.000,B 0.000,C 90.000,E1 292.025} C_DIS
LIN {X 0.074,Y -649.310,Z 1026.420,A 0.000,B 0.000,C 90.000,E1 291.535} C_DIS
LIN {X 0.157,Y -649.019,Z 1026.418,A 0.000,B 0.000,C 90.000,E1 291.280} C_DIS
LIN {X 0.083,Y -647.996,Z 1026.416,A 0.000,B 0.000,C 90.000,E1 290.791} C_DIS
LIN {X -0.070,Y -647.176,Z 1026.414,A 0.000,B 0.000,C 90.000,E1 290.556} C_DIS
LIN {X -0.033,Y -646.588,Z 1026.414,A 0.000,B 0.000,C 90.000,E1 290.429} C_DIS
LIN {X -0.152,Y -644.322,Z 1026.411,A 0.000,B 0.000,C 90.000,E1 290.066} C_DIS
LIN {X -0.122,Y -643.362,Z 1026.411,A 0.000,B 0.000,C 90.000,E1 289.939} C_DIS
LIN {X 0.063,Y -640.372,Z 1026.409,A 0.000,B 0.000,C 90.000,E1 289.685} C_DIS
LIN {X 0.005,Y -638.050,Z 1026.408,A 0.000,B 0.000,C 90.000,E1 289.450} C_DIS
LIN {X 0.024,Y -636.375,Z 1026.407,A 0.000,B 0.000,C 90.000,E1 289.322} C_DIS
LIN {X -0.247,Y -629.344,Z 1026.405,A 0.000,B 0.000,C 90.000,E1 288.960} C_DIS
LIN {X 0.115,Y -620.601,Z 1026.403,A 0.000,B 0.000,C 90.000,E1 288.544} C_DIS
LIN {X -0.130,Y -611.484,Z 1026.401,A 0.000,B 0.000,C 90.000,E1 288.236} C_DIS
LIN {X 0.214,Y -608.098,Z 1026.401,A 0.000,B 0.000,C 90.000,E1 288.055} C_DIS
LIN {X 0.271,Y -606.695,Z 1026.400,A 0.000,B 0.000,C 90.000,E1 288.000} C_DIS
LIN {X 0.224,Y -606.618,Z 1026.400,A 0.000,B 0.000,C 90.000,E1 288.000} C_DIS
LIN {X -0.184,Y -608.214,Z 1026.399,A 0.000,B 0.000,C 90.000,E1 287.819} C_DIS
LIN {X 0.252,Y -613.323,Z 1026.396,A 0.000,B 0.000,C 90.000,E1 287.275} C_DIS
LIN {X -0.101,Y -618.031,Z 1026.393,A 0.000,B 0.000,C 90.000,E1 286.804} C_DIS
LIN {X 0.182,Y -622.791,Z 1026.390,A 0.000,B 0.000,C 90.000,E1 286.134} C_DIS
LIN {X 0.332,Y -626.717,Z 1026.386,A 0.000,B 0.000,C 90.000,E1 285.481} C_DIS
LIN {X -0.057,Y -628.714,Z 1026.384,A 0.000,B 0.000,C 90.000,E1 285.134} C_DIS
LIN {X 0.322,Y -631.150,Z 1026.381,A 0.000,B 0.000,C 90.000,E1 284.592} C_DIS
LIN {X -0.246,Y -633.869,Z 1026.377,A 0.000,B 0.000,C 90.000,E1 283.883} C_DIS
LIN {X 0.006,Y -635.218,Z 1026.374,A 0.000,B 0.000,C 90.000,E1 283.355} C_DIS
LIN {X 0.095,Y -636.463,Z 1026.370,A 0.000,B 0.000,C 90.000,E1 282.591} C_DIS
LIN {X -0.253,Y -636.903,Z 1026.367,A 0.000,B 0.000,C 90.000,E1 282.119} C_DIS
LIN {X 0.022,Y -636.895,Z 1026.365,A 0.000,B 0.000,C 90.000,E1 281.591} C_DIS
LIN {X -0.279,Y -636.745,Z 1026.363,A 0.000,B 0.000,C 90.000,E1 281.366} C_DIS
LIN {X -0.002,Y -636.163,Z 1026.360,A 0.000,B 0.000,C 90.000,E1 280.838} C_DIS
LIN {X 0.269,Y -635.113,Z 1026.357,A 0.000,B 0.000,C 90.000,E1 280.310} C_DIS
LIN {X -0.204,Y -633.687,Z 1026.355,A 0.000,B 0.000,C 90.000,E1 279.849} C_DIS
LIN {X 0.234,Y -632.800,Z 1026.353,A 0.000,B 0.000,C 90.000,E1 279.557} C_DIS
LIN {X -0.247,Y -630.541,Z 1026.350,A 0.000,B 0.000,C 90.000,E1 279.095} C_DIS
LIN {X -0.024,Y -627.748,Z 1026.348,A 0.000,B 0.000,C 90.000,E1 278.568} C_DIS
LIN {X 0.084,Y -624.408,Z 1026.345,A 0.000,B 0.000,C 90.000,E1 278.049} C_DIS
LIN {X -0.138,Y -622.299,Z 1026.343,A 0.000,B 0.000,C 90.000,E1 277.814} C_DIS
LIN {X -0.195,Y -616.267,Z 1026.340,A 0.000,B 0.000,C 90.000,E1 277.182} C_DIS
LIN {X -0.323,Y -615.046,Z 1026.339,A 0.000,B 0.000,C 90.000,E1 277.068} C_DIS
LIN {X 0.096,Y -610.623,Z 1026.337,A 0.000,B 0.000,C 90.000,E1 276.663} C_DIS
LIN {X 0.205,Y -607.870,Z 1026.336,A 0.000,B 0.000,C 90.000,E1 276.429} C_DIS
LIN {X 0.219,Y -600.068,Z 1026.333,A 0.000,B 0.000,C 90.000,E1 275.910} C_DIS
LIN {X -0.104,Y -593.380,Z 1026.331,A 0.000,B 0.000,C 90.000,E1 275.568} C_DIS
LIN {X 0.282,Y -587.824,Z 1026.329,A 0.000,B 0.000,C 90.000,E1 275.277} C_DIS
LIN {X 0.073,Y -585.741,Z 1026.329,A 0.000,B 0.000,C 90.000,E1 275.220} C_DIS
LIN {X -0.023,Y -579.717,Z 1026.328,A 0.000,B 0.000,C 90.000,E1 275.049} C_DIS
LIN {X -0.161,Y -573.746,Z 1026.327,A 0.000,B 0.000,C 90.000,E1 274.935} C_DIS
LIN {X 0.032,Y -571.499,Z 1026.327,A 0.000,B 0.000,C 90.000,E1 274.878} C_DIS
LIN {X 0.063,Y -566.420,Z 1026.327,A 0.000,B 0.000,C 90.000,E1 274.821} C_DIS
LIN {X 0.009,Y -544.002,Z 1026.327,A 0.000,B 0.000,C 90.000,E1 274.821} C_DIS
LIN {X -0.127,Y -543.198,Z 1026.325,A 0.000,B 0.000,C 90.000,E1 274.531} C_DIS
LIN {X -0.029,Y -542.694,Z 1026.324,A 0.000,B 0.000,C 90.000,E1 274.245} C_DIS
LIN {X 0.176,Y -541.183,Z 1026.314,A 0.000,B 0.000,C 90.000,E1 272.522} C_DIS
LIN {X -0.218,Y -540.366,Z 1026.305,A 0.000,B 0.000,C 90.000,E1 270.859} C_DIS
LIN {X -0.135,Y -539.727,Z 1026.298,A 0.000,B 0.000,C 90.000,E1 269.714} C_DIS
LIN {X -0.051,Y -538.703,Z 1026.291,A 0.000,B 0.000,C 90.000,E1 268.282} C_DIS
LIN {X 0.061,Y -537.410,Z 1026.281,A 0.000,B 0.000,C 90.000,E1 266.560} C_DIS
LIN {X 0.187,Y -535.678,Z 1026.268,A 0.000,B 0.000,C 90.000,E1 264.261} C_DIS
LIN {X -0.231,Y -534.608,Z 1026.260,A 0.000,B 0.000,C 90.000,E1 262.875} C_DIS
LIN {X -0.141,Y -533.222,Z 1026.252,A 0.000,B 0.000,C 90.000,E1 261.432} C_DIS
LIN {X -0.004,Y -532.314,Z 1026.248,A 0.000,B 0.000,C 90.000,E1 260.557} C_DIS
LIN {X -0.218,Y -529.066,Z 1026.232,A 0.000,B 0.000,C 90.000,E1 257.701} C_DIS
LIN {X 0.053,Y -527.485,Z 1026.224,A 0.000,B 0.000,C 90.000,E1 256.228} C_DIS
LIN {X -0.217,Y -525.904,Z 1026.216,A 0.000,B 0.000,C 90.000,E1 254.810} C_DIS
LIN {X -0.219,Y -523.705,Z 1026.204,A 0.000,B 0.000,C 90.000,E1 252.779} C_DIS
LIN {X 0.234,Y -522.139,Z 1026.196,A 0.000,B 0.000,C 90.000,E1 251.275} C_DIS
LIN {X -0.186,Y -519.888,Z 1026.186,A 0.000,B 0.000,C 90.000,E1 249.571} C_DIS
LIN {X 0.010,Y -517.562,Z 1026.177,A 0.000,B 0.000,C 90.000,E1 247.794} C_DIS
LIN {X -0.262,Y -515.634,Z 1026.169,A 0.000,B 0.000,C 90.000,E1 246.357} C_DIS
LIN {X -0.008,Y -513.979,Z 1026.162,A 0.000,B 0.000,C 90.000,E1 245.153} C_DIS
LIN {X -0.002,Y -512.161,Z 1026.155,A 0.000,B 0.000,C 90.000,E1 243.973} C_DIS
LIN {X 0.065,Y -509.785,Z 1026.147,A 0.000,B 0.000,C 90.000,E1 242.487} C_DIS
LIN {X 0.088,Y -507.269,Z 1026.139,A 0.000,B 0.000,C 90.000,E1 241.001} C_DIS
LIN {X 0.180,Y -504.057,Z 1026.129,A 0.000,B 0.000,C 90.000,E1 239.203} C_DIS
LIN {X -0.100,Y -501.274,Z 1026.121,A 0.000,B 0.000,C 90.000,E1 237.740} C_DIS
LIN {X 0.235,Y -498.873,Z 1026.114,A 0.000,B 0.000,C 90.000,E1 236.501} C_DIS
LIN {X 0.257,Y -496.956,Z 1026.109,A 0.000,B 0.000,C 90.000,E1 235.595} C_DIS
LIN {X 0.259,Y -494.915,Z 1026.104,A 0.000,B 0.000,C 90.000,E1 234.689} C_DIS
LIN {X -0.211,Y -490.714,Z 1026.094,A 0.000,B 0.000,C 90.000,E1 232.924} C_DIS
LIN {X -0.011,Y -487.034,Z 1026.085,A 0.000,B 0.000,C 90.000,E1 231.376} C_DIS
LIN {X -0.120,Y -481.479,Z 1026.072,A 0.000,B 0.000,C 90.000,E1 228.933} C_DIS
LIN {X -0.026,Y -475.414,Z 1026.056,A 0.000,B 0.000,C 90.000,E1 226.134} C_DIS
LIN {X -0.184,Y -472.196,Z 1026.048,A 0.000,B 0.000,C 90.000,E1 224.595} C_DIS
LIN {X 0.015,Y -468.306,Z 1026.037,A 0.000,B 0.000,C 90.000,E1 222.690} C_DIS
LIN {X 0.154,Y -464.497,Z 1026.027,A 0.000,B 0.000,C 90.000,E1 220.782} C_DIS
LIN {X -0.241,Y -461.902,Z 1026.020,A 0.000,B 0.000,C 90.000,E1 219.564} C_DIS
LIN {X -0.065,Y -459.735,Z 1026.014,A 0.000,B 0.000,C 90.000,E1 218.588} C_DIS
LIN {X -0.268,Y -454.698,Z 1026.002,A 0.000,B 0.000,C 90.000,E1 216.377} C_DIS
LIN {X 0.057,Y -450.502,Z 1025.991,A 0.000,B 0.000,C 90.000,E1 214.405} C_DIS
LIN {X -0.051,Y -447.033,Z 1025.982,A 0.000,B 0.000,C 90.000,E1 212.801} C_DIS
LIN {X -0.043,Y -442.809,Z 1025.971,A 0.000,B 0.000,C 90.000,E1 210.846} C_DIS
LIN {X -0.017,Y -439.203,Z 1025.962,A 0.000,B 0.000,C 90.000,E1 209.205} C_DIS
LIN {X -0.088,Y -436.177,Z 1025.955,A 0.000,B 0.000,C 90.000,E1 207.897} C_DIS
LIN {X -0.004,Y -431.625,Z 1025.944,A 0.000,B 0.000,C 90.000,E1 205.899} C_DIS
LIN {X -0.036,Y -426.425,Z 1025.931,A 0.000,B 0.000,C 90.000,E1 203.567} C_DIS
LIN {X -0.146,Y -421.502,Z 1025.918,A 0.000,B 0.000,C 90.000,E1 201.227} C_DIS
LIN {X -0.211,Y -415.886,Z 1025.901,A 0.000,B 0.000,C 90.000,E1 198.181} C_DIS
LIN {X -0.065,Y -409.226,Z 1025.876,A 0.000,B 0.000,C 90.000,E1 193.703} C_DIS
LIN {X 0.116,Y -407.219,Z 1025.867,A 0.000,B 0.000,C 90.000,E1 191.951} C_DIS
LIN {X -0.158,Y -406.539,Z 1025.861,A 0.000,B 0.000,C 90.000,E1 190.950} C_DIS
LIN {X -0.058,Y -406.612,Z 1025.859,A 0.000,B 0.000,C 90.000,E1 190.602} C_DIS
LIN {X -0.046,Y -406.538,Z 1025.857,A 0.000,B 0.000,C 90.000,E1 190.254} C_DIS
LIN {X -0.017,Y -407.270,Z 1025.853,A 0.000,B 0.000,C 90.000,E1 189.557} C_DIS
LIN {X 0.023,Y -407.362,Z 1025.852,A 0.000,B 0.000,C 90.000,E1 189.378} C_DIS
LIN {X 0.089,Y -409.491,Z 1025.848,A 0.000,B 0.000,C 90.000,E1 188.624} C_DIS
LIN {X 0.109,Y -410.858,Z 1025.846,A 0.000,B 0.000,C 90.000,E1 188.276} C_DIS
LIN {X 0.150,Y -414.509,Z 1025.842,A 0.000,B 0.000,C 90.000,E1 187.587} C_DIS
LIN {X 0.191,Y -416.654,Z 1025.840,A 0.000,B 0.000,C 90.000,E1 187.239} C_DIS
LIN {X -0.011,Y -422.518,Z 1025.836,A 0.000,B 0.000,C 90.000,E1 186.429} C_DIS
LIN {X 0.122,Y -435.252,Z 1025.827,A 0.000,B 0.000,C 90.000,E1 184.759} C_DIS
LIN {X 0.058,Y -444.350,Z 1025.820,A 0.000,B 0.000,C 90.000,E1 183.612} C_DIS
LIN {X 0.207,Y -454.608,Z 1025.813,A 0.000,B 0.000,C 90.000,E1 182.293} C_DIS
LIN {X -0.043,Y -463.440,Z 1025.807,A 0.000,B 0.000,C 90.000,E1 181.203} C_DIS
LIN {X -0.073,Y -472.886,Z 1025.800,A 0.000,B 0.000,C 90.000,E1 179.943} C_DIS
LIN {X -0.239,Y -479.584,Z 1025.794,A 0.000,B 0.000,C 90.000,E1 179.026} C_DIS
LIN {X -0.168,Y -487.246,Z 1025.788,A 0.000,B 0.000,C 90.000,E1 177.936} C_DIS
LIN {X 0.016,Y -494.638,Z 1025.783,A 0.000,B 0.000,C 90.000,E1 176.846} C_DIS
LIN {X -0.014,Y -502.435,Z 1025.776,A 0.000,B 0.000,C 90.000,E1 175.641} C_DIS
LIN {X 0.173,Y -508.231,Z 1025.771,A 0.000,B 0.000,C 90.000,E1 174.723} C_DIS
LIN {X -0.224,Y -516.256,Z 1025.764,A 0.000,B 0.000,C 90.000,E1 173.451} C_DIS
LIN {X 0.099,Y -524.744,Z 1025.755,A 0.000,B 0.000,C 90.000,E1 171.951} C_DIS
LIN {X -0.078,Y -528.883,Z 1025.751,A 0.000,B 0.000,C 90.000,E1 171.254} C_DIS
LIN {X -0.018,Y -535.439,Z 1025.745,A 0.000,B 0.000,C 90.000,E1 170.095} C_DIS
LIN {X -0.046,Y -542.864,Z 1025.738,A 0.000,B 0.000,C 90.000,E1 168.814} C_DIS
LIN {X -0.119,Y -550.872,Z 1025.730,A 0.000,B 0.000,C 90.000,E1 167.409} C_DIS
LIN {X -0.313,Y -555.415,Z 1025.725,A 0.000,B 0.000,C 90.000,E1 166.589} C_DIS
LIN {X -0.042,Y -562.848,Z 1025.718,A 0.000,B 0.000,C 90.000,E1 165.172} C_DIS
LIN {X 0.191,Y -568.739,Z 1025.712,A 0.000,B 0.000,C 90.000,E1 164.047} C_DIS
LIN {X -0.242,Y -575.678,Z 1025.704,A 0.000,B 0.000,C 90.000,E1 162.725} C_DIS
LIN {X 0.228,Y -578.940,Z 1025.700,A 0.000,B 0.000,C 90.000,E1 162.000} C_DIS
LIN {X -0.165,Y -583.325,Z 1025.695,A 0.000,B 0.000,C 90.000,E1 161.094} C_DIS
LIN {X -0.034,Y -587.910,Z 1025.689,A 0.000,B 0.000,C 90.000,E1 160.007} C_DIS
LIN {X -0.191,Y -592.389,Z 1025.683,A 0.000,B 0.000,C 90.000,E1 158.954} C_DIS
LIN {X 0.274,Y -596.603,Z 1025.677,A 0.000,B 0.000,C 90.000,E1 157.847} C_DIS
LIN {X 0.244,Y -600.426,Z 1025.671,A 0.000,B 0.000,C 90.000,E1 156.794} C_DIS
LIN {X -0.221,Y -603.114,Z 1025.667,A 0.000,B 0.000,C 90.000,E1 156.049} C_DIS
LIN {X 0.078,Y -606.502,Z 1025.661,A 0.000,B 0.000,C 90.000,E1 154.973} C_DIS
LIN {X -0.162,Y -610.440,Z 1025.654,A 0.000,B 0.000,C 90.000,E1 153.691} C_DIS
LIN {X 0.239,Y -613.365,Z 1025.648,A 0.000,B 0.000,C 90.000,E1 152.615} C_DIS
LIN {X 0.102,Y -616.813,Z 1025.641,A 0.000,B 0.000,C 90.000,E1 151.335} C_DIS
LIN {X 0.057,Y -621.405,Z 1025.631,A 0.000,B 0.000,C 90.000,E1 149.537} C_DIS
LIN {X 0.133,Y -624.618,Z 1025.624,A 0.000,B 0.000,C 90.000,E1 148.250} C_DIS
LIN {X -0.071,Y -627.179,Z 1025.618,A 0.000,B 0.000,C 90.000,E1 147.248} C_DIS
LIN {X -0.069,Y -630.924,Z 1025.610,A 0.000,B 0.000,C 90.000,E1 145.722} C_DIS
LIN {X 0.009,Y -634.597,Z 1025.601,A 0.000,B 0.000,C 90.000,E1 144.196} C_DIS
LIN {X -0.249,Y -637.043,Z 1025.596,A 0.000,B 0.000,C 90.000,E1 143.210} C_DIS
LIN {X -0.200,Y -640.689,Z 1025.587,A 0.000,B 0.000,C 90.000,E1 141.698} C_DIS
LIN {X -0.088,Y -643.702,Z 1025.580,A 0.000,B 0.000,C 90.000,E1 140.436} C_DIS
LIN {X -0.069,Y -647.856,Z 1025.571,A 0.000,B 0.000,C 90.000,E1 138.690} C_DIS
LIN {X -0.058,Y -653.307,Z 1025.558,A 0.000,B 0.000,C 90.000,E1 136.458} C_DIS
LIN {X -0.357,Y -658.613,Z 1025.547,A 0.000,B 0.000,C 90.000,E1 134.514} C_DIS
LIN {X -0.039,Y -664.470,Z 1025.536,A 0.000,B 0.000,C 90.000,E1 132.528} C_DIS
LIN {X -0.023,Y -667.355,Z 1025.531,A 0.000,B 0.000,C 90.000,E1 131.553} C_DIS
LIN {X -0.469,Y -670.284,Z 1025.526,A 0.000,B 0.000,C 90.000,E1 130.620} C_DIS
LIN {X 0.051,Y -672.356,Z 1025.521,A 0.000,B 0.000,C 90.000,E1 129.850} C_DIS
LIN {X -0.247,Y -675.742,Z 1025.515,A 0.000,B 0.000,C 90.000,E1 128.669} C_DIS
LIN {X 0.026,Y -678.334,Z 1025.509,A 0.000,B 0.000,C 90.000,E1 127.684} C_DIS
LIN {X -0.019,Y -682.174,Z 1025.501,A 0.000,B 0.000,C 90.000,E1 126.251} C_DIS
LIN {X 0.376,Y -685.376,Z 1025.495,A 0.000,B 0.000,C 90.000,E1 125.025} C_DIS
LIN {X 0.048,Y -689.034,Z 1025.487,A 0.000,B 0.000,C 90.000,E1 123.627} C_DIS
LIN {X -0.017,Y -692.585,Z 1025.479,A 0.000,B 0.000,C 90.000,E1 122.212} C_DIS
LIN {X 0.103,Y -694.896,Z 1025.474,A 0.000,B 0.000,C 90.000,E1 121.258} C_DIS
LIN {X -0.110,Y -696.938,Z 1025.469,A 0.000,B 0.000,C 90.000,E1 120.335} C_DIS
LIN {X -0.294,Y -698.685,Z 1025.463,A 0.000,B 0.000,C 90.000,E1 119.411} C_DIS
LIN {X -0.112,Y -699.746,Z 1025.459,A 0.000,B 0.000,C 90.000,E1 118.693} C_DIS
LIN {X -0.267,Y -700.947,Z 1025.454,A 0.000,B 0.000,C 90.000,E1 117.769} C_DIS
LIN {X -0.183,Y -702.196,Z 1025.446,A 0.000,B 0.000,C 90.000,E1 116.360} C_DIS
LIN {X -0.001,Y -703.029,Z 1025.441,A 0.000,B 0.000,C 90.000,E1 115.412} C_DIS
LIN {X -0.090,Y -703.480,Z 1025.437,A 0.000,B 0.000,C 90.000,E1 114.719} C_DIS
LIN {X -0.167,Y -703.470,Z 1025.435,A 0.000,B 0.000,C 90.000,E1 114.259} C_DIS
LIN {X -0.174,Y -703.286,Z 1025.433,A 0.000,B 0.000,C 90.000,E1 114.027} C_DIS
LIN {X 0.386,Y -702.462,Z 1025.431,A 0.000,B 0.000,C 90.000,E1 113.515} C_DIS
LIN {X -0.261,Y -701.564,Z 1025.430,A 0.000,B 0.000,C 90.000,E1 113.334} C_DIS
LIN {X 0.281,Y -698.969,Z 1025.427,A 0.000,B 0.000,C 90.000,E1 112.823} C_DIS
LIN {X 0.142,Y -698.049,Z 1025.426,A 0.000,B 0.000,C 90.000,E1 112.717} C_DIS
LIN {X 0.273,Y -696.679,Z 1025.426,A 0.000,B 0.000,C 90.000,E1 112.589} C_DIS
LIN {X 0.115,Y -690.109,Z 1025.423,A 0.000,B 0.000,C 90.000,E1 112.206} C_DIS
LIN {X -0.326,Y -688.031,Z 1025.423,A 0.000,B 0.000,C 90.000,E1 112.153} C_DIS
LIN {X 0.129,Y -685.266,Z 1025.422,A 0.000,B 0.000,C 90.000,E1 112.025} C_DIS
LIN {X 0.097,Y -682.502,Z 1025.422,A 0.000,B 0.000,C 90.000,E1 111.972} C_DIS
LIN {X -0.081,Y -675.222,Z 1025.422,A 0.000,B 0.000,C 90.000,E1 111.897} C_DIS
LIN {X -0.123,Y -613.753,Z 1025.422,A 0.000,B 0.000,C 90.000,E1 111.897} C_DIS
LIN {X -0.105,Y -611.580,Z 1025.421,A 0.000,B 0.000,C 90.000,E1 111.844} C_DIS
LIN {X 0.198,Y -604.926,Z 1025.420,A 0.000,B 0.000,C 90.000,E1 111.589} C_DIS
LIN {X -0.238,Y -599.059,Z 1025.419,A 0.000,B 0.000,C 90.000,E1 111.354} C_DIS
LIN {X 0.269,Y -593.521,Z 1025.417,A 0.000,B 0.000,C 90.000,E1 110.972} C_DIS
LIN {X -0.196,Y -587.933,Z 1025.414,A 0.000,B 0.000,C 90.000,E1 110.610} C_DIS
LIN {X 0.064,Y -577.608,Z 1025.410,A 0.000,B 0.000,C 90.000,E1 109.704} C_DIS
LIN {X -0.153,Y -571.441,Z 1025.407,A 0.000,B 0.000,C 90.000,E1 109.268} C_DIS
LIN {X 0.029,Y -569.817,Z 1025.406,A 0.000,B 0.000,C 90.000,E1 109.141} C_DIS
LIN {X 0.008,Y -561.388,Z 1025.404,A 0.000,B 0.000,C 90.000,E1 108.671} C_DIS
LIN {X 0.218,Y -554.789,Z 1025.402,A 0.000,B 0.000,C 90.000,E1 108.308} C_DIS
LIN {X 0.106,Y -549.620,Z 1025.400,A 0.000,B 0.000,C 90.000,E1 108.000} C_DIS
LIN {X 0.177,Y -548.159,Z 1025.399,A 0.000,B 0.000,C 90.000,E1 107.819} C_DIS
LIN {X 0.135,Y -548.132,Z 1025.399,A 0.000,B 0.000,C 90.000,E1 107.819} C_DIS
LIN {X 0.141,Y -547.763,Z 1025.397,A 0.000,B 0.000,C 90.000,E1 107.528} C_DIS
LIN {X 0.067,Y -548.715,Z 1025.386,A 0.000,B 0.000,C 90.000,E1 105.426} C_DIS
LIN {X 0.112,Y -551.036,Z 1025.365,A 0.000,B 0.000,C 90.000,E1 101.771} C_DIS
LIN {X -0.018,Y -553.573,Z 1025.352,A 0.000,B 0.000,C 90.000,E1 99.265} C_DIS
LIN {X -0.040,Y -555.206,Z 1025.344,A 0.000,B 0.000,C 90.000,E1 97.871} C_DIS
LIN {X -0.116,Y -556.774,Z 1025.336,A 0.000,B 0.000,C 90.000,E1 96.486} C_DIS
LIN {X -0.222,Y -558.113,Z 1025.328,A 0.000,B 0.000,C 90.000,E1 95.106} C_DIS
LIN {X 0.055,Y -558.758,Z 1025.324,A 0.000,B 0.000,C 90.000,E1 94.245} C_DIS
LIN {X -0.013,Y -559.607,Z 1025.316,A 0.000,B 0.000,C 90.000,E1 92.865} C_DIS
LIN {X -0.195,Y -560.153,Z 1025.310,A 0.000,B 0.000,C 90.000,E1 91.776} C_DIS
LIN {X -0.197,Y -560.815,Z 1025.301,A 0.000,B 0.000,C 90.000,E1 90.115} C_DIS
LIN {X -0.068,Y -561.498,Z 1025.290,A 0.000,B 0.000,C 90.000,E1 88.165} C_DIS
LIN {X -0.117,Y -561.936,Z 1025.282,A 0.000,B 0.000,C 90.000,E1 86.788} C_DIS
LIN {X -0.167,Y -562.245,Z 1025.274,A 0.000,B 0.000,C 90.000,E1 85.412} C_DIS
LIN {X -0.033,Y -562.639,Z 1025.265,A 0.000,B 0.000,C 90.000,E1 83.742} C_DIS
LIN {X 0.013,Y -563.245,Z 1025.251,A 0.000,B 0.000,C 90.000,E1 81.254} C_DIS
LIN {X -0.162,Y -563.872,Z 1025.241,A 0.000,B 0.000,C 90.000,E1 79.342} C_DIS
LIN {X 0.044,Y -564.911,Z 1025.229,A 0.000,B 0.000,C 90.000,E1 77.117} C_DIS
LIN {X 0.238,Y -566.112,Z 1025.218,A 0.000,B 0.000,C 90.000,E1 75.172} C_DIS
LIN {X 0.005,Y -567.977,Z 1025.204,A 0.000,B 0.000,C 90.000,E1 72.725} C_DIS
LIN {X -0.128,Y -569.189,Z 1025.195,A 0.000,B 0.000,C 90.000,E1 71.094} C_DIS
LIN {X -0.042,Y -570.448,Z 1025.186,A 0.000,B 0.000,C 90.000,E1 69.444} C_DIS
LIN {X -0.107,Y -571.698,Z 1025.175,A 0.000,B 0.000,C 90.000,E1 67.539} C_DIS
LIN {X -0.293,Y -572.583,Z 1025.166,A 0.000,B 0.000,C 90.000,E1 65.921} C_DIS
LIN {X -0.230,Y -573.377,Z 1025.157,A 0.000,B 0.000,C 90.000,E1 64.280} C_DIS
LIN {X -0.061,Y -574.199,Z 1025.146,A 0.000,B 0.000,C 90.000,E1 62.359} C_DIS
LIN {X 0.083,Y -574.621,Z 1025.140,A 0.000,B 0.000,C 90.000,E1 61.257} C_DIS
LIN {X -0.144,Y -575.087,Z 1025.133,A 0.000,B 0.000,C 90.000,E1 59.921} C_DIS
LIN {X 0.138,Y -575.520,Z 1025.125,A 0.000,B 0.000,C 90.000,E1 58.535} C_DIS
LIN {X 0.214,Y -576.121,Z 1025.115,A 0.000,B 0.000,C 90.000,E1 56.628} C_DIS
LIN {X -0.002,Y -576.328,Z 1025.106,A 0.000,B 0.000,C 90.000,E1 55.022} C_DIS
LIN {X 0.125,Y -576.369,Z 1025.101,A 0.000,B 0.000,C 90.000,E1 54.196} C_DIS
LIN {X 0.090,Y -576.191,Z 1025.094,A 0.000,B 0.000,C 90.000,E1 52.844} C_DIS
LIN {X 0.096,Y -576.097,Z 1025.089,A 0.000,B 0.000,C 90.000,E1 52.029} C_DIS
LIN {X 0.043,Y -575.458,Z 1025.082,A 0.000,B 0.000,C 90.000,E1 50.678} C_DIS
LIN {X -0.258,Y -574.942,Z 1025.076,A 0.000,B 0.000,C 90.000,E1 49.622} C_DIS
LIN {X -0.046,Y -573.957,Z 1025.068,A 0.000,B 0.000,C 90.000,E1 48.243} C_DIS
LIN {X 0.019,Y -572.979,Z 1025.062,A 0.000,B 0.000,C 90.000,E1 47.148} C_DIS
LIN {X -0.048,Y -572.112,Z 1025.057,A 0.000,B 0.000,C 90.000,E1 46.338} C_DIS
LIN {X 0.288,Y -571.061,Z 1025.053,A 0.000,B 0.000,C 90.000,E1 45.486} C_DIS
LIN {X 0.203,Y -569.778,Z 1025.048,A 0.000,B 0.000,C 90.000,E1 44.676} C_DIS
LIN {X -0.203,Y -567.871,Z 1025.042,A 0.000,B 0.000,C 90.000,E1 43.623} C_DIS
LIN {X 0.086,Y -566.227,Z 1025.038,A 0.000,B 0.000,C 90.000,E1 42.771} C_DIS
LIN {X -0.061,Y -564.368,Z 1025.033,A 0.000,B 0.000,C 90.000,E1 41.962} C_DIS
LIN {X 0.139,Y -563.037,Z 1025.030,A 0.000,B 0.000,C 90.000,E1 41.391} C_DIS
LIN {X 0.374,Y -560.735,Z 1025.026,A 0.000,B 0.000,C 90.000,E1 40.539} C_DIS
LIN {X 0.218,Y -558.196,Z 1025.021,A 0.000,B 0.000,C 90.000,E1 39.725} C_DIS
LIN {X -0.042,Y -556.309,Z 1025.018,A 0.000,B 0.000,C 90.000,E1 39.197} C_DIS
LIN {X -0.242,Y -553.244,Z 1025.013,A 0.000,B 0.000,C 90.000,E1 38.382} C_DIS
LIN {X -0.038,Y -549.928,Z 1025.009,A 0.000,B 0.000,C 90.000,E1 37.523} C_DIS
LIN {X 0.129,Y -546.180,Z 1025.004,A 0.000,B 0.000,C 90.000,E1 36.664} C_DIS
LIN {X 0.070,Y -542.873,Z 1025.000,A 0.000,B 0.000,C 90.000,E1 35.964} C_DIS
LIN {X 0.007,Y -537.919,Z 1024.994,A 0.000,B 0.000,C 90.000,E1 34.978} C_DIS
LIN {X 0.029,Y -533.373,Z 1024.990,A 0.000,B 0.000,C 90.000,E1 34.119} C_DIS
LIN {X -0.145,Y -529.358,Z 1024.986,A 0.000,B 0.000,C 90.000,E1 33.420} C_DIS
LIN {X -0.075,Y -524.189,Z 1024.981,A 0.000,B 0.000,C 90.000,E1 32.546} C_DIS
LIN {X -0.002,Y -520.543,Z 1024.978,A 0.000,B 0.000,C 90.000,E1 31.957} C_DIS
LIN {X -0.124,Y -516.661,Z 1024.974,A 0.000,B 0.000,C 90.000,E1 31.386} C_DIS
LIN {X 0.246,Y -510.275,Z 1024.969,A 0.000,B 0.000,C 90.000,E1 30.463} C_DIS
LIN {X 0.219,Y -505.676,Z 1024.966,A 0.000,B 0.000,C 90.000,E1 29.873} C_DIS
LIN {X 0.161,Y -500.728,Z 1024.963,A 0.000,B 0.000,C 90.000,E1 29.283} C_DIS
LIN {X -0.012,Y -494.094,Z 1024.959,A 0.000,B 0.000,C 90.000,E1 28.565} C_DIS
LIN {X 0.203,Y -489.982,Z 1024.956,A 0.000,B 0.000,C 90.000,E1 28.103} C_DIS
LIN {X 0.228,Y -482.950,Z 1024.952,A 0.000,B 0.000,C 90.000,E1 27.385} C_DIS
LIN {X -0.240,Y -474.404,Z 1024.948,A 0.000,B 0.000,C 90.000,E1 26.616} C_DIS
LIN {X 0.067,Y -467.044,Z 1024.944,A 0.000,B 0.000,C 90.000,E1 25.899} C_DIS
LIN {X 0.237,Y -459.597,Z 1024.940,A 0.000,B 0.000,C 90.000,E1 25.207} C_DIS
LIN {X -0.040,Y -448.944,Z 1024.935,A 0.000,B 0.000,C 90.000,E1 24.335} C_DIS
LIN {X -0.017,Y -432.462,Z 1024.927,A 0.000,B 0.000,C 90.000,E1 22.898} C_DIS
LIN {X 0.159,Y -417.678,Z 1024.919,A 0.000,B 0.000,C 90.000,E1 21.461} C_DIS
LIN {X -0.065,Y -402.101,Z 1024.910,A 0.000,B 0.000,C 90.000,E1 19.812} C_DIS
LIN {X -0.147,Y -398.676,Z 1024.908,A 0.000,B 0.000,C 90.000,E1 19.396} C_DIS
LIN {X -0.113,Y -396.575,Z 1024.906,A 0.000,B 0.000,C 90.000,E1 19.087} C_DIS
LIN {X 0.009,Y -392.769,Z 1024.902,A 0.000,B 0.000,C 90.000,E1 18.417} C_DIS
LIN {X -0.169,Y -391.965,Z 1024.901,A 0.000,B 0.000,C 90.000,E1 18.181} C_DIS
LIN {X -0.144,Y -391.597,Z 1024.900,A 0.000,B 0.000,C 90.000,E1 18.000} C_DIS
LIN {X -0.045,Y -391.111,Z 1024.897,A 0.000,B 0.000,C 90.000,E1 17.457} C_DIS
LIN {X 0.004,Y -391.187,Z 1024.894,A 0.000,B 0.000,C 90.000,E1 16.858} C_DIS
LIN {X 0.075,Y -392.321,Z 1024.886,A 0.000,B 0.000,C 90.000,E1 15.426} C_DIS
LIN {X 0.058,Y -397.006,Z 1024.864,A 0.000,B 0.000,C 90.000,E1 11.535} C_DIS
LIN {X -0.182,Y -405.269,Z 1024.837,A 0.000,B 0.000,C 90.000,E1 6.663} C_DIS
LIN {X 0.184,Y -411.152,Z 1024.822,A 0.000,B 0.000,C 90.000,E1 3.841} C_DIS
LIN {X 0.189,Y -413.496,Z 1024.816,A 0.000,B 0.000,C 90.000,E1 2.808} C_DIS
LIN {X 0.193,Y -414.943,Z 1024.813,A 0.000,B 0.000,C 90.000,E1 2.293} C_DIS
LIN {X -0.193,Y -416.935,Z 1024.810,A 0.000,B 0.000,C 90.000,E1 1.833} C_DIS
LIN {X -0.177,Y -418.050,Z 1024.809,A 0.000,B 0.000,C 90.000,E1 1.661} C_DIS
LIN {X -0.125,Y -422.187,Z 1024.806,A 0.000,B 0.000,C 90.000,E1 1.146} C_DIS
LIN {X -0.092,Y -423.984,Z 1024.805,A 0.000,B 0.000,C 90.000,E1 0.974} C_DIS
LIN {X -0.056,Y -427.730,Z 1024.804,A 0.000,B 0.000,C 90.000,E1 0.688} C_DIS
LIN {X 0.162,Y -433.315,Z 1024.802,A 0.000,B 0.000,C 90.000,E1 0.344} C_DIS
LIN {X 0.134,Y -449.401,Z 1024.797,A 0.000,B 0.000,C 90.000,E1 359.370} C_DIS
LIN {X -0.026,Y -466.039,Z 1024.791,A 0.000,B 0.000,C 90.000,E1 358.396} C_DIS
LIN {X -0.114,Y -480.653,Z 1024.786,A 0.000,B 0.000,C 90.000,E1 357.535} C_DIS
LIN {X -0.066,Y -492.137,Z 1024.782,A 0.000,B 0.000,C 90.000,E1 356.846} C_DIS
LIN {X 0.058,Y -500.171,Z 1024.780,A 0.000,B 0.000,C 90.000,E1 356.331} C_DIS
LIN {X -0.243,Y -511.230,Z 1024.776,A 0.000,B 0.000,C 90.000,E1 355.641} C_DIS
LIN {X 0.029,Y -518.858,Z 1024.773,A 0.000,B 0.000,C 90.000,E1 355.065} C_DIS
LIN {X 0.030,Y -524.767,Z 1024.770,A 0.000,B 0.000,C 90.000,E1 354.609} C_DIS
LIN {X -0.100,Y -530.504,Z 1024.767,A 0.000,B 0.000,C 90.000,E1 354.147} C_DIS
LIN {X 0.112,Y -536.165,Z 1024.765,A 0.000,B 0.000,C 90.000,E1 353.628} C_DIS
LIN {X 0.227,Y -541.595,Z 1024.762,A 0.000,B 0.000,C 90.000,E1 353.109} C_DIS
LIN {X 0.085,Y -546.757,Z 1024.759,A 0.000,B 0.000,C 90.000,E1 352.591} C_DIS
LIN {X 0.074,Y -552.786,Z 1024.755,A 0.000,B 0.000,C 90.000,E1 351.894} C_DIS
LIN {X 0.229,Y -557.311,Z 1024.752,A 0.000,B 0.000,C 90.000,E1 351.319} C_DIS
LIN {X -0.300,Y -562.215,Z 1024.748,A 0.000,B 0.000,C 90.000,E1 350.679} C_DIS
LIN {X 0.011,Y -565.901,Z 1024.745,A 0.000,B 0.000,C 90.000,E1 350.095} C_DIS
LIN {X -0.075,Y -573.212,Z 1024.738,A 0.000,B 0.000,C 90.000,E1 348.870} C_DIS
LIN {X 0.089,Y -576.834,Z 1024.734,A 0.000,B 0.000,C 90.000,E1 348.173} C_DIS
LIN {X -0.162,Y -580.177,Z 1024.731,A 0.000,B 0.000,C 90.000,E1 347.521} C_DIS
LIN {X 0.194,Y -585.172,Z 1024.725,A 0.000,B 0.000,C 90.000,E1 346.408} C_DIS
LIN {X 0.037,Y -589.848,Z 1024.719,A 0.000,B 0.000,C 90.000,E1 345.353} C_DIS
LIN {X 0.084,Y -594.302,Z 1024.713,A 0.000,B 0.000,C 90.000,E1 344.283} C_DIS
LIN {X 0.365,Y -598.590,Z 1024.707,A 0.000,B 0.000,C 90.000,E1 343.196} C_DIS
LIN {X -0.038,Y -602.635,Z 1024.701,A 0.000,B 0.000,C 90.000,E1 342.181} C_DIS
LIN {X 0.093,Y -607.350,Z 1024.694,A 0.000,B 0.000,C 90.000,E1 340.859} C_DIS
LIN {X 0.257,Y -609.940,Z 1024.689,A 0.000,B 0.000,C 90.000,E1 340.061} C_DIS
LIN {X 0.187,Y -613.128,Z 1024.684,A 0.000,B 0.000,C 90.000,E1 339.028} C_DIS
LIN {X -0.191,Y -616.103,Z 1024.678,A 0.000,B 0.000,C 90.000,E1 338.028} C_DIS
LIN {X 0.049,Y -618.906,Z 1024.672,A 0.000,B 0.000,C 90.000,E1 336.975} C_DIS
LIN {X 0.319,Y -622.167,Z 1024.665,A 0.000,B 0.000,C 90.000,E1 335.665} C_DIS
LIN {X 0.069,Y -625.010,Z 1024.658,A 0.000,B 0.000,C 90.000,E1 334.409} C_DIS
LIN {X 0.151,Y -628.021,Z 1024.649,A 0.000,B 0.000,C 90.000,E1 332.871} C_DIS
LIN {X 0.214,Y -629.403,Z 1024.645,A 0.000,B 0.000,C 90.000,E1 332.103} C_DIS
LIN {X 0.090,Y -631.377,Z 1024.638,A 0.000,B 0.000,C 90.000,E1 330.845} C_DIS
LIN {X 0.009,Y -633.189,Z 1024.631,A 0.000,B 0.000,C 90.000,E1 329.587} C_DIS
LIN {X -0.047,Y -634.653,Z 1024.624,A 0.000,B 0.000,C 90.000,E1 328.329} C_DIS
LIN {X 0.122,Y -636.328,Z 1024.614,A 0.000,B 0.000,C 90.000,E1 326.548} C_DIS
LIN {X 0.055,Y -637.097,Z 1024.609,A 0.000,B 0.000,C 90.000,E1 325.548} C_DIS
LIN {X -0.177,Y -637.587,Z 1024.603,A 0.000,B 0.000,C 90.000,E1 324.562} C_DIS
LIN {X -0.022,Y -637.927,Z 1024.598,A 0.000,B 0.000,C 90.000,E1 323.543} C_DIS
LIN {X 0.152,Y -638.200,Z 1024.591,A 0.000,B 0.000,C 90.000,E1 322.271} C_DIS
LIN {X -0.291,Y -638.488,Z 1024.582,A 0.000,B 0.000,C 90.000,E1 320.803} C_DIS
LIN {X -0.319,Y -638.972,Z 1024.574,A 0.000,B 0.000,C 90.000,E1 319.299} C_DIS
LIN {X 0.268,Y -639.424,Z 1024.568,A 0.000,B 0.000,C 90.000,E1 318.243} C_DIS
LIN {X -0.229,Y -639.856,Z 1024.560,A 0.000,B 0.000,C 90.000,E1 316.782} C_DIS
LIN {X 0.080,Y -640.540,Z 1024.550,A 0.000,B 0.000,C 90.000,E1 315.000} C_DIS
LIN {X 0.048,Y -641.167,Z 1024.542,A 0.000,B 0.000,C 90.000,E1 313.500} C_DIS
LIN {X 0.112,Y -641.769,Z 1024.535,A 0.000,B 0.000,C 90.000,E1 312.243} C_DIS
LIN {X 0.089,Y -642.279,Z 1024.526,A 0.000,B 0.000,C 90.000,E1 310.744} C_DIS
LIN {X 0.217,Y -642.589,Z 1024.520,A 0.000,B 0.000,C 90.000,E1 309.483} C_DIS
LIN {X -0.143,Y -643.032,Z 1024.511,A 0.000,B 0.000,C 90.000,E1 308.016} C_DIS
LIN {X 0.012,Y -643.195,Z 1024.503,A 0.000,B 0.000,C 90.000,E1 306.503} C_DIS
LIN {X -0.211,Y -643.560,Z 1024.495,A 0.000,B 0.000,C 90.000,E1 305.025} C_DIS
LIN {X 0.146,Y -644.452,Z 1024.481,A 0.000,B 0.000,C 90.000,E1 302.498} C_DIS
LIN {X -0.280,Y -646.528,Z 1024.465,A 0.000,B 0.000,C 90.000,E1 299.795} C_DIS
LIN {X 0.225,Y -648.866,Z 1024.453,A 0.000,B 0.000,C 90.000,E1 297.513} C_DIS
LIN {X 0.109,Y -650.107,Z 1024.446,A 0.000,B 0.000,C 90.000,E1 296.283} C_DIS
LIN {X 0.115,Y -650.766,Z 1024.442,A 0.000,B 0.000,C 90.000,E1 295.540} C_DIS
LIN {X -0.084,Y -651.278,Z 1024.437,A 0.000,B 0.000,C 90.000,E1 294.567} C_DIS
LIN {X -0.059,Y -651.437,Z 1024.432,A 0.000,B 0.000,C 90.000,E1 293.823} C_DIS
LIN {X -0.090,Y -651.337,Z 1024.426,A 0.000,B 0.000,C 90.000,E1 292.589} C_DIS
LIN {X -0.056,Y -651.094,Z 1024.421,A 0.000,B 0.000,C 90.000,E1 291.844} C_DIS
LIN {X -0.116,Y -650.508,Z 1024.419,A 0.000,B 0.000,C 90.000,E1 291.354} C_DIS
LIN {X 0.055,Y -649.519,Z 1024.416,A 0.000,B 0.000,C 90.000,E1 290.844} C_DIS
LIN {X -0.094,Y -648.883,Z 1024.415,A 0.000,B 0.000,C 90.000,E1 290.610} C_DIS
LIN {X -0.017,Y -647.465,Z 1024.413,A 0.000,B 0.000,C 90.000,E1 290.355} C_DIS
LIN {X -0.135,Y -645.164,Z 1024.411,A 0.000,B 0.000,C 90.000,E1 289.993} C_DIS
LIN {X -0.103,Y -644.074,Z 1024.410,A 0.000,B 0.000,C 90.000,E1 289.866} C_DIS
LIN {X -0.014,Y -639.434,Z 1024.408,A 0.000,B 0.000,C 90.000,E1 289.504} C_DIS
LIN {X 0.021,Y -638.376,Z 1024.408,A 0.000,B 0.000,C 90.000,E1 289.396} C_DIS
LIN {X 0.069,Y -636.541,Z 1024.407,A 0.000,B 0.000,C 90.000,E1 289.268} C_DIS
LIN {X -0.111,Y -629.402,Z 1024.405,A 0.000,B 0.000,C 90.000,E1 288.906} C_DIS
LIN {X -0.186,Y -620.704,Z 1024.403,A 0.000,B 0.000,C 90.000,E1 288.544} C_DIS
LIN {X 0.167,Y -611.724,Z 1024.401,A 0.000,B 0.000,C 90.000,E1 288.181} C_DIS
LIN {X -0.247,Y -609.850,Z 1024.401,A 0.000,B 0.000,C 90.000,E1 288.127} C_DIS
LIN {X -0.110,Y -609.787,Z 1024.401,A 0.000,B 0.000,C 90.000,E1 288.109} C_DIS
LIN {X 0.288,Y -619.101,Z 1024.395,A 0.000,B 0.000,C 90.000,E1 287.040} C_DIS
LIN {X 0.010,Y -623.236,Z 1024.392,A 0.000,B 0.000,C 90.000,E1 286.551} C_DIS
LIN {X 0.195,Y -625.662,Z 1024.390,A 0.000,B 0.000,C 90.000,E1 286.150} C_DIS
LIN {X 0.131,Y -628.143,Z 1024.388,A 0.000,B 0.000,C 90.000,E1 285.788} C_DIS
LIN {X -0.281,Y -631.504,Z 1024.384,A 0.000,B 0.000,C 90.000,E1 285.190} C_DIS
LIN {X 0.140,Y -632.670,Z 1024.383,A 0.000,B 0.000,C 90.000,E1 284.898} C_DIS
LIN {X 0.362,Y -635.640,Z 1024.379,A 0.000,B 0.000,C 90.000,E1 284.120} C_DIS
LIN {X 0.183,Y -636.557,Z 1024.377,A 0.000,B 0.000,C 90.000,E1 283.883} C_DIS
LIN {X 0.285,Y -638.169,Z 1024.373,A 0.000,B 0.000,C 90.000,E1 283.119} C_DIS
LIN {X -0.053,Y -639.079,Z 1024.370,A 0.000,B 0.000,C 90.000,E1 282.647} C_DIS
LIN {X 0.238,Y -639.394,Z 1024.368,A 0.000,B 0.000,C 90.000,E1 282.119} C_DIS
LIN {X 0.072,Y -639.434,Z 1024.366,A 0.000,B 0.000,C 90.000,E1 281.883} C_DIS
LIN {X 0.238,Y -639.223,Z 1024.363,A 0.000,B 0.000,C 90.000,E1 281.366} C_DIS
LIN {X -0.094,Y -638.706,Z 1024.360,A 0.000,B 0.000,C 90.000,E1 280.894} C_DIS
LIN {X 0.193,Y -637.766,Z 1024.358,A 0.000,B 0.000,C 90.000,E1 280.366} C_DIS
LIN {X -0.267,Y -636.415,Z 1024.355,A 0.000,B 0.000,C 90.000,E1 279.905} C_DIS
LIN {X 0.183,Y -635.641,Z 1024.354,A 0.000,B 0.000,C 90.000,E1 279.613} C_DIS
LIN {X -0.283,Y -633.651,Z 1024.351,A 0.000,B 0.000,C 90.000,E1 279.151} C_DIS
LIN {X -0.036,Y -631.245,Z 1024.348,A 0.000,B 0.000,C 90.000,E1 278.624} C_DIS
LIN {X -0.181,Y -630.539,Z 1024.347,A 0.000,B 0.000,C 90.000,E1 278.511} C_DIS
LIN {X -0.053,Y -627.066,Z 1024.344,A 0.000,B 0.000,C 90.000,E1 277.992} C_DIS
LIN {X 0.053,Y -622.935,Z 1024.342,A 0.000,B 0.000,C 90.000,E1 277.473} C_DIS
LIN {X 0.246,Y -617.993,Z 1024.339,A 0.000,B 0.000,C 90.000,E1 276.947} C_DIS
LIN {X 0.020,Y -615.342,Z 1024.337,A 0.000,B 0.000,C 90.000,E1 276.720} C_DIS
LIN {X -0.063,Y -611.000,Z 1024.335,A 0.000,B 0.000,C 90.000,E1 276.372} C_DIS
LIN {X 0.050,Y -606.485,Z 1024.334,A 0.000,B 0.000,C 90.000,E1 276.030} C_DIS
LIN {X -0.120,Y -601.788,Z 1024.332,A 0.000,B 0.000,C 90.000,E1 275.739} C_DIS
LIN {X 0.223,Y -595.367,Z 1024.330,A 0.000,B 0.000,C 90.000,E1 275.334} C_DIS
LIN {X -0.117,Y -593.752,Z 1024.329,A 0.000,B 0.000,C 90.000,E1 275.277} C_DIS
LIN {X 0.251,Y -586.387,Z 1024.328,A 0.000,B 0.000,C 90.000,E1 274.935} C_DIS
LIN {X 0.187,Y -580.642,Z 1024.327,A 0.000,B 0.000,C 90.000,E1 274.759} C_DIS
LIN {X 0.205,Y -578.493,Z 1024.326,A 0.000,B 0.000,C 90.000,E1 274.702} C_DIS
LIN {X -0.129,Y -573.835,Z 1024.326,A 0.000,B 0.000,C 90.000,E1 274.645} C_DIS
LIN {X 0.092,Y -571.635,Z 1024.326,A 0.000,B 0.000,C 90.000,E1 274.588} C_DIS
LIN {X 0.073,Y -566.949,Z 1024.325,A 0.000,B 0.000,C 90.000,E1 274.531} C_DIS
LIN {X -0.053,Y -566.165,Z 1024.325,A 0.000,B 0.000,C 90.000,E1 274.531} C_DIS
LIN {X -0.176,Y -559.715,Z 1024.325,A 0.000,B 0.000,C 90.000,E1 274.531} C_DIS
LIN {X -0.211,Y -543.898,Z 1024.325,A 0.000,B 0.000,C 90.000,E1 274.531} C_DIS
LIN {X -0.215,Y -543.355,Z 1024.324,A 0.000,B 0.000,C 90.000,E1 274.359} C_DIS
LIN {X 0.132,Y -542.583,Z 1024.322,A 0.000,B 0.000,C 90.000,E1 273.898} C_DIS
LIN {X 0.182,Y -542.061,Z 1024.319,A 0.000,B 0.000,C 90.000,E1 273.326} C_DIS
LIN {X 0.236,Y -541.710,Z 1024.317,A 0.000,B 0.000,C 90.000,E1 273.037} C_DIS
LIN {X -0.109,Y -540.472,Z 1024.304,A 0.000,B 0.000,C 90.000,E1 270.802} C_DIS
LIN {X -0.025,Y -539.837,Z 1024.298,A 0.000,B 0.000,C 90.000,E1 269.656} C_DIS
LIN {X 0.060,Y -538.820,Z 1024.290,A 0.000,B 0.000,C 90.000,E1 268.224} C_DIS
LIN {X 0.174,Y -537.517,Z 1024.281,A 0.000,B 0.000,C 90.000,E1 266.502} C_DIS
LIN {X -0.231,Y -535.799,Z 1024.268,A 0.000,B 0.000,C 90.000,E1 264.261} C_DIS
LIN {X -0.116,Y -534.691,Z 1024.260,A 0.000,B 0.000,C 90.000,E1 262.818} C_DIS
LIN {X 0.004,Y -533.616,Z 1024.254,A 0.000,B 0.000,C 90.000,E1 261.659} C_DIS
LIN {X 0.111,Y -532.401,Z 1024.247,A 0.000,B 0.000,C 90.000,E1 260.500} C_DIS
LIN {X -0.106,Y -529.167,Z 1024.231,A 0.000,B 0.000,C 90.000,E1 257.645} C_DIS
LIN {X 0.164,Y -527.593,Z 1024.223,A 0.000,B 0.000,C 90.000,E1 256.172} C_DIS
LIN {X -0.125,Y -526.335,Z 1024.217,A 0.000,B 0.000,C 90.000,E1 255.046} C_DIS
LIN {X -0.113,Y -523.781,Z 1024.204,A 0.000,B 0.000,C 90.000,E1 252.725} C_DIS
LIN {X -0.157,Y -522.220,Z 1024.196,A 0.000,B 0.000,C 90.000,E1 251.275} C_DIS
LIN {X -0.087,Y -519.976,Z 1024.186,A 0.000,B 0.000,C 90.000,E1 249.518} C_DIS
LIN {X 0.159,Y -518.050,Z 1024.178,A 0.000,B 0.000,C 90.000,E1 248.028} C_DIS
LIN {X -0.170,Y -515.709,Z 1024.168,A 0.000,B 0.000,C 90.000,E1 246.305} C_DIS
LIN {X 0.080,Y -514.025,Z 1024.162,A 0.000,B 0.000,C 90.000,E1 245.101} C_DIS
LIN {X -0.154,Y -512.247,Z 1024.155,A 0.000,B 0.000,C 90.000,E1 243.948} C_DIS
LIN {X -0.309,Y -509.871,Z 1024.147,A 0.000,B 0.000,C 90.000,E1 242.487} C_DIS
LIN {X -0.037,Y -507.357,Z 1024.139,A 0.000,B 0.000,C 90.000,E1 240.973} C_DIS
LIN {X -0.185,Y -504.178,Z 1024.129,A 0.000,B 0.000,C 90.000,E1 239.203} C_DIS
LIN {X 0.231,Y -501.346,Z 1024.120,A 0.000,B 0.000,C 90.000,E1 237.661} C_DIS
LIN {X 0.005,Y -499.592,Z 1024.115,A 0.000,B 0.000,C 90.000,E1 236.786} C_DIS
LIN {X -0.099,Y -497.002,Z 1024.109,A 0.000,B 0.000,C 90.000,E1 235.595} C_DIS
LIN {X -0.096,Y -494.961,Z 1024.104,A 0.000,B 0.000,C 90.000,E1 234.689} C_DIS
LIN {X 0.126,Y -490.712,Z 1024.094,A 0.000,B 0.000,C 90.000,E1 232.844} C_DIS
LIN {X 0.021,Y -487.033,Z 1024.085,A 0.000,B 0.000,C 90.000,E1 231.331} C_DIS
LIN {X 0.216,Y -481.457,Z 1024.072,A 0.000,B 0.000,C 90.000,E1 228.852} C_DIS
LIN {X 0.308,Y -475.397,Z 1024.056,A 0.000,B 0.000,C 90.000,E1 226.053} C_DIS
LIN {X 0.147,Y -472.207,Z 1024.047,A 0.000,B 0.000,C 90.000,E1 224.514} C_DIS
LIN {X -0.318,Y -468.289,Z 1024.037,A 0.000,B 0.000,C 90.000,E1 222.690} C_DIS
LIN {X -0.177,Y -464.461,Z 1024.026,A 0.000,B 0.000,C 90.000,E1 220.782} C_DIS
LIN {X 0.079,Y -461.851,Z 1024.019,A 0.000,B 0.000,C 90.000,E1 219.483} C_DIS
LIN {X -0.006,Y -458.943,Z 1024.012,A 0.000,B 0.000,C 90.000,E1 218.222} C_DIS
LIN {X 0.041,Y -454.630,Z 1024.002,A 0.000,B 0.000,C 90.000,E1 216.297} C_DIS
LIN {X 0.019,Y -451.157,Z 1023.993,A 0.000,B 0.000,C 90.000,E1 214.692} C_DIS
LIN {X 0.001,Y -446.975,Z 1023.982,A 0.000,B 0.000,C 90.000,E1 212.752} C_DIS
LIN {X 0.016,Y -442.737,Z 1023.971,A 0.000,B 0.000,C 90.000,E1 210.797} C_DIS
LIN {X 0.001,Y -439.869,Z 1023.964,A 0.000,B 0.000,C 90.000,E1 209.489} C_DIS
LIN {X 0.154,Y -436.866,Z 1023.957,A 0.000,B 0.000,C 90.000,E1 208.153} C_DIS
LIN {X 0.061,Y -432.341,Z 1023.946,A 0.000,B 0.000,C 90.000,E1 206.181} C_DIS
